SPLINE
SPL {X  -154.371, Y  +335.471, Z    +0.000, E1   +73.016, E3 +26676.206}
SPL {X  -149.938, Y  +321.685, Z    +0.000, E1   +73.398, E3 +26680.901}
SPL {X  -145.016, Y  +309.920, Z    +0.000, E1   +73.647, E3 +26685.422}
SPL {X  -139.138, Y  +298.522, Z    +0.000, E1   +74.138, E3 +26687.438}
SPL {X  -135.697, Y  +292.747, Z    +0.000, E1   +74.259, E3 +26689.439}
SPL {X  -132.590, Y  +287.964, Z    +0.000, E1   +73.910, E3 +26694.468}
SPL {X  -129.541, Y  +283.606, Z    +0.000, E1   +73.551, E3 +26699.108}
SPL {X  -126.457, Y  +279.493, Z    +0.000, E1   +73.175, E3 +26703.507}
SPL {X  -122.770, Y  +274.912, Z    +0.000, E1   +72.712, E3 +26708.362}
SPL {X  -118.941, Y  +270.496, Z    +0.000, E1   +72.188, E3 +26712.950}
SPL {X   -74.907, Y  +236.129, Z    +0.000, E1   +61.720, E3 +26791.563}
ENDSPLINE

SPLINE
SPL {X   -94.059, Y  +248.080, Z    +0.000, E1   +58.275, E3 +27013.256}
SPL {X  -136.558, Y  +294.141, Z    +0.000, E1   +54.887, E3 +27057.111}
SPL {X  -151.843, Y  +327.098, Z    +0.000, E1   +44.118, E3 +27066.470}
SPL {X  -157.484, Y  +349.293, Z    +0.000, E1   +30.654, E3 +27069.510}
SPL {X  -159.556, Y  +365.719, Z    +0.000, E1   +15.845, E3 +27070.702}
SPL {X  -159.982, Y  +375.924, Z    +0.000, E1    +4.476, E3 +27071.004}
SPL {X  -159.990, Y  +379.531, Z    +0.000, E1    -0.039, E3 +27071.031}
SPL {X  -159.990, Y  +382.420, Z    +0.000, E1    -7.600, E3 +27071.059}
SPL {X  -159.990, Y  +386.504, Z    +0.000, E1   -19.860, E3 +27071.165}
SPL {X  -159.990, Y  +392.530, Z    +0.000, E1   -36.133, E3 +27071.480}
SPL {X  -159.990, Y  +400.492, Z    +0.000, E1   -51.837, E3 +27072.133}
SPL {X  -159.990, Y  +409.662, Z    +0.000, E1   -61.705, E3 +27073.244}
SPL {X  -159.990, Y  +434.697, Z    +0.000, E1   -71.504, E3 +27078.264}
SPL {X  -159.990, Y  +521.523, Z    +0.000, E1   -76.035, E3 +27104.544}
SPL {X  -154.459, Y  +718.205, Z    +0.000, E1   -76.329, E3 +27186.340}
SPL {X  -151.356, Y  +728.349, Z    +0.000, E1   -76.056, E3 +27194.555}
SPL {X  -148.399, Y  +736.287, Z    +0.000, E1   -75.788, E3 +27201.434}
SPL {X  -144.005, Y  +746.209, Z    +0.000, E1   -75.396, E3 +27210.550}
SPL {X  -138.117, Y  +757.250, Z    +0.000, E1   -74.803, E3 +27221.440}
SPL {X  -133.491, Y  +764.686, Z    +0.000, E1   -74.276, E3 +27229.181}
SPL {X  -128.839, Y  +771.354, Z    +0.000, E1   -73.759, E3 +27236.199}
SPL {X  -123.568, Y  +778.125, Z    +0.000, E1   -73.105, E3 +27243.371}
SPL {X  -118.985, Y  +783.455, Z    +0.000, E1   -72.490, E3 +27248.879}
SPL {X   -72.391, Y  +819.176, Z    +0.000, E1   -59.867, E3 +27345.565}
ENDSPLINE

SPLINE
SPL {X   -92.809, Y  +806.820, Z    +0.000, E1   -56.994, E3 +27538.360}
SPL {X  -120.521, Y  +781.721, Z    +0.000, E1   -56.766, E3 +27574.459}
SPL {X  -148.710, Y  +735.509, Z    +0.000, E1   -46.282, E3 +27595.740}
SPL {X  -157.559, Y  +704.285, Z    +0.000, E1   -29.037, E3 +27601.069}
SPL {X  -159.430, Y  +689.871, Z    +0.000, E1   -16.582, E3 +27602.219}
SPL {X  -159.960, Y  +679.609, Z    +0.000, E1    -6.021, E3 +27602.602}
SPL {X  -159.990, Y  +674.508, Z    +0.000, E1    -0.018, E3 +27602.661}
SPL {X  -159.990, Y  +672.787, Z    +0.000, E1    +4.022, E3 +27602.673}
SPL {X  -159.990, Y  +669.267, Z    +0.000, E1   +13.665, E3 +27602.743}
SPL {X  -159.990, Y  +663.438, Z    +0.000, E1   +29.379, E3 +27603.014}
SPL {X  -159.990, Y  +655.264, Z    +0.000, E1   +47.291, E3 +27603.631}
SPL {X  -159.990, Y  +645.368, Z    +0.000, E1   +59.257, E3 +27604.874}
SPL {X  -159.990, Y  +624.023, Z    +0.000, E1   +69.513, E3 +27608.999}
SPL {X  -159.990, Y  +543.075, Z    +0.000, E1   +75.590, E3 +27632.647}
SPL {X  -156.121, Y  +342.530, Z    +0.000, E1   +75.868, E3 +27719.293}
SPL {X  -153.865, Y  +333.657, Z    +0.000, E1   +75.438, E3 +27728.897}
ENDSPLINE

SPLINE
SPL {X  -159.644, Y  +366.989, Z    +0.000, E1   +72.058, E3 +27744.424}
ENDSPLINE

SPLINE
SPL {X  -156.933, Y  +346.374, Z    +0.000, E1   +72.645, E3 +27752.313}
SPL {X  -151.144, Y  +325.039, Z    +0.000, E1   +73.323, E3 +27758.993}
SPL {X  -145.016, Y  +309.920, Z    +0.000, E1   +73.647, E3 +27764.787}
SPL {X  -136.944, Y  +294.777, Z    +0.000, E1   +74.219, E3 +27768.088}
SPL {X  -132.590, Y  +287.964, Z    +0.000, E1   +73.910, E3 +27773.833}
SPL {X  -129.541, Y  +283.606, Z    +0.000, E1   +73.551, E3 +27778.473}
SPL {X  -125.403, Y  +278.147, Z    +0.000, E1   +73.063, E3 +27784.280}
SPL {X  -121.908, Y  +273.889, Z    +0.000, E1   +72.578, E3 +27788.827}
SPL {X  -118.941, Y  +270.496, Z    +0.000, E1   +72.188, E3 +27792.315}
SPL {X   -74.907, Y  +236.129, Z    +0.000, E1   +61.720, E3 +27870.928}
ENDSPLINE

SPLINE
SPL {X   -94.059, Y  +248.080, Z    +0.000, E1   +58.275, E3 +28092.621}
SPL {X  -136.558, Y  +294.141, Z    +0.000, E1   +54.887, E3 +28136.476}
SPL {X  -151.843, Y  +327.098, Z    +0.000, E1   +44.118, E3 +28145.835}
SPL {X  -157.484, Y  +349.293, Z    +0.000, E1   +30.654, E3 +28148.875}
SPL {X  -159.556, Y  +365.719, Z    +0.000, E1   +15.845, E3 +28150.067}
SPL {X  -159.982, Y  +375.924, Z    +0.000, E1    +4.476, E3 +28150.369}
SPL {X  -159.990, Y  +379.531, Z    +0.000, E1    -0.039, E3 +28150.396}
SPL {X  -159.990, Y  +382.420, Z    +0.000, E1    -7.600, E3 +28150.424}
SPL {X  -159.990, Y  +386.504, Z    +0.000, E1   -19.860, E3 +28150.530}
SPL {X  -159.990, Y  +392.530, Z    +0.000, E1   -36.133, E3 +28150.845}
SPL {X  -159.990, Y  +400.492, Z    +0.000, E1   -51.837, E3 +28151.498}
SPL {X  -159.990, Y  +409.662, Z    +0.000, E1   -61.705, E3 +28152.609}
SPL {X  -159.990, Y  +434.697, Z    +0.000, E1   -71.504, E3 +28157.629}
SPL {X  -159.990, Y  +521.523, Z    +0.000, E1   -76.035, E3 +28183.909}
SPL {X  -154.459, Y  +718.205, Z    +0.000, E1   -76.329, E3 +28265.705}
SPL {X  -151.356, Y  +728.349, Z    +0.000, E1   -76.056, E3 +28273.920}
SPL {X  -148.399, Y  +736.287, Z    +0.000, E1   -75.788, E3 +28280.799}
SPL {X  -144.005, Y  +746.209, Z    +0.000, E1   -75.396, E3 +28289.915}
SPL {X  -138.117, Y  +757.250, Z    +0.000, E1   -74.803, E3 +28300.805}
SPL {X  -133.491, Y  +764.686, Z    +0.000, E1   -74.276, E3 +28308.546}
SPL {X  -130.530, Y  +769.013, Z    +0.000, E1   -73.929, E3 +28313.128}
SPL {X  -127.734, Y  +772.837, Z    +0.000, E1   -73.601, E3 +28317.180}
SPL {X  -124.765, Y  +776.652, Z    +0.000, E1   -73.233, E3 +28321.214}
SPL {X  -121.376, Y  +780.734, Z    +0.000, E1   -72.804, E3 +28325.476}
SPL {X  -118.281, Y  +784.233, Z    +0.000, E1   -72.371, E3 +28329.044}
SPL {X   -72.391, Y  +819.176, Z    +0.000, E1   -59.867, E3 +28424.930}
ENDSPLINE

SPLINE
SPL {X   -92.809, Y  +806.820, Z    +0.000, E1   -56.994, E3 +28617.725}
SPL {X  -120.521, Y  +781.721, Z    +0.000, E1   -56.766, E3 +28653.824}
SPL {X  -148.710, Y  +735.509, Z    +0.000, E1   -46.282, E3 +28675.105}
SPL {X  -157.559, Y  +704.285, Z    +0.000, E1   -29.037, E3 +28680.434}
SPL {X  -159.430, Y  +689.871, Z    +0.000, E1   -16.582, E3 +28681.584}
SPL {X  -159.960, Y  +679.609, Z    +0.000, E1    -6.021, E3 +28681.968}
SPL {X  -159.990, Y  +674.508, Z    +0.000, E1    -0.018, E3 +28682.026}
SPL {X  -159.990, Y  +672.787, Z    +0.000, E1    +4.022, E3 +28682.038}
SPL {X  -159.990, Y  +669.267, Z    +0.000, E1   +13.665, E3 +28682.108}
SPL {X  -159.990, Y  +665.069, Z    +0.000, E1   +25.376, E3 +28682.280}
SPL {X  -159.990, Y  +657.821, Z    +0.000, E1   +42.408, E3 +28682.782}
SPL {X  -159.990, Y  +645.368, Z    +0.000, E1   +59.257, E3 +28684.239}
SPL {X  -159.990, Y  +624.023, Z    +0.000, E1   +69.513, E3 +28688.364}
SPL {X  -159.990, Y  +543.075, Z    +0.000, E1   +75.590, E3 +28712.012}
SPL {X  -156.121, Y  +342.530, Z    +0.000, E1   +75.868, E3 +28798.658}
SPL {X  -153.498, Y  +332.386, Z    +0.000, E1   +75.628, E3 +28806.663}
ENDSPLINE

SPLINE
SPL {X  -155.252, Y  +338.851, Z    +0.000, E1   +74.632, E3 +28814.041}
SPL {X  -159.644, Y  +366.989, Z    +0.000, E1   +72.058, E3 +28823.789}
ENDSPLINE

SPLINE
SPL {X  -156.933, Y  +346.374, Z    +0.000, E1   +72.645, E3 +28831.678}
SPL {X  -151.144, Y  +325.039, Z    +0.000, E1   +73.323, E3 +28838.358}
SPL {X  -146.668, Y  +313.584, Z    +0.000, E1   +73.560, E3 +28842.840}
SPL {X  -141.230, Y  +302.327, Z    +0.000, E1   +73.933, E3 +28845.811}
SPL {X  -135.697, Y  +292.747, Z    +0.000, E1   +74.259, E3 +28848.170}
SPL {X  -132.590, Y  +287.964, Z    +0.000, E1   +73.910, E3 +28853.198}
SPL {X  -129.541, Y  +283.606, Z    +0.000, E1   +73.551, E3 +28857.838}
SPL {X  -125.403, Y  +278.147, Z    +0.000, E1   +73.063, E3 +28863.645}
SPL {X  -121.908, Y  +273.889, Z    +0.000, E1   +72.578, E3 +28868.192}
SPL {X  -118.941, Y  +270.496, Z    +0.000, E1   +72.188, E3 +28871.680}
SPL {X   -74.907, Y  +236.129, Z    +0.000, E1   +61.720, E3 +28950.293}
SPL {X   -72.759, Y  +235.012, Z    +0.000, E1   +56.036, E3 +29121.971}
ENDSPLINE

SPLINE
SPL {X  -123.257, Y  +275.497, Z    +0.000, E1   +57.800, E3 +29205.847}
SPL {X  -149.689, Y  +321.019, Z    +0.000, E1   +46.817, E3 +29223.947}
SPL {X  -157.484, Y  +349.293, Z    +0.000, E1   +30.654, E3 +29228.240}
SPL {X  -159.556, Y  +365.719, Z    +0.000, E1   +15.845, E3 +29229.432}
SPL {X  -159.982, Y  +375.924, Z    +0.000, E1    +4.476, E3 +29229.734}
SPL {X  -159.990, Y  +379.531, Z    +0.000, E1    -0.039, E3 +29229.761}
SPL {X  -159.990, Y  +382.420, Z    +0.000, E1    -7.600, E3 +29229.789}
SPL {X  -159.990, Y  +387.978, Z    +0.000, E1   -23.882, E3 +29229.958}
SPL {X  -159.990, Y  +396.850, Z    +0.000, E1   -45.459, E3 +29230.545}
SPL {X  -159.990, Y  +409.662, Z    +0.000, E1   -61.705, E3 +29231.974}
SPL {X  -159.990, Y  +426.583, Z    +0.000, E1   -69.729, E3 +29235.088}
SPL {X  -159.990, Y  +451.842, Z    +0.000, E1   -73.935, E3 +29241.015}
SPL {X  -159.990, Y  +521.523, Z    +0.000, E1   -76.035, E3 +29263.275}
SPL {X  -154.459, Y  +718.205, Z    +0.000, E1   -76.329, E3 +29345.070}
SPL {X  -151.356, Y  +728.349, Z    +0.000, E1   -76.056, E3 +29353.285}
SPL {X  -148.399, Y  +736.287, Z    +0.000, E1   -75.788, E3 +29360.164}
SPL {X  -144.005, Y  +746.209, Z    +0.000, E1   -75.396, E3 +29369.280}
SPL {X  -138.117, Y  +757.250, Z    +0.000, E1   -74.803, E3 +29380.170}
SPL {X  -133.491, Y  +764.686, Z    +0.000, E1   -74.276, E3 +29387.911}
SPL {X  -130.530, Y  +769.013, Z    +0.000, E1   -73.929, E3 +29392.493}
SPL {X  -127.734, Y  +772.837, Z    +0.000, E1   -73.601, E3 +29396.545}
SPL {X  -123.568, Y  +778.125, Z    +0.000, E1   -73.105, E3 +29402.101}
SPL {X  -118.985, Y  +783.455, Z    +0.000, E1   -72.490, E3 +29407.609}
SPL {X   -72.391, Y  +819.176, Z    +0.000, E1   -59.867, E3 +29504.295}
ENDSPLINE

SPLINE
SPL {X  -116.241, Y  +786.431, Z    +0.000, E1   -57.120, E3 +29728.737}
SPL {X  -148.710, Y  +735.509, Z    +0.000, E1   -46.282, E3 +29754.470}
SPL {X  -156.039, Y  +711.834, Z    +0.000, E1   -34.227, E3 +29758.955}
SPL {X  -158.281, Y  +699.823, Z    +0.000, E1   -25.469, E3 +29760.246}
SPL {X  -159.709, Y  +685.986, Z    +0.000, E1   -12.810, E3 +29761.131}
SPL {X  -159.990, Y  +674.648, Z    +0.000, E1    -0.349, E3 +29761.390}
SPL {X  -159.990, Y  +672.787, Z    +0.000, E1    +4.022, E3 +29761.403}
SPL {X  -159.990, Y  +669.267, Z    +0.000, E1   +13.665, E3 +29761.473}
SPL {X  -159.990, Y  +665.069, Z    +0.000, E1   +25.376, E3 +29761.645}
SPL {X  -159.990, Y  +657.821, Z    +0.000, E1   +42.408, E3 +29762.147}
SPL {X  -159.990, Y  +645.368, Z    +0.000, E1   +59.257, E3 +29763.604}
SPL {X  -159.990, Y  +624.023, Z    +0.000, E1   +69.513, E3 +29767.729}
SPL {X  -159.990, Y  +543.075, Z    +0.000, E1   +75.590, E3 +29791.377}
SPL {X  -156.121, Y  +342.530, Z    +0.000, E1   +75.868, E3 +29878.023}
SPL {X  -153.498, Y  +332.386, Z    +0.000, E1   +75.628, E3 +29886.028}
ENDSPLINE

SPLINE
SPL {X  -155.252, Y  +338.851, Z    +0.000, E1   +74.632, E3 +29893.406}
SPL {X  -159.103, Y  +360.678, Z    +0.000, E1   +72.233, E3 +29905.731}
ENDSPLINE

SPLINE
SPL {X  -154.371, Y  +335.471, Z    +0.000, E1   +73.016, E3 +29914.302}
SPL {X  -149.938, Y  +321.685, Z    +0.000, E1   +73.398, E3 +29918.996}
SPL {X  -145.016, Y  +309.920, Z    +0.000, E1   +73.647, E3 +29923.517}
SPL {X  -139.138, Y  +298.522, Z    +0.000, E1   +74.138, E3 +29925.533}
SPL {X  -135.697, Y  +292.747, Z    +0.000, E1   +74.259, E3 +29927.535}
SPL {X  -132.590, Y  +287.964, Z    +0.000, E1   +73.910, E3 +29932.563}
SPL {X  -129.541, Y  +283.606, Z    +0.000, E1   +73.551, E3 +29937.203}
SPL {X  -126.457, Y  +279.493, Z    +0.000, E1   +73.175, E3 +29941.602}
SPL {X  -122.770, Y  +274.912, Z    +0.000, E1   +72.712, E3 +29946.458}
SPL {X  -119.156, Y  +270.736, Z    +0.000, E1   +72.213, E3 +29950.807}
SPL {X  -117.531, Y  +268.949, Z    +0.000, E1   +71.964, E3 +29952.622}
SPL {X   -74.907, Y  +236.129, Z    +0.000, E1   +61.720, E3 +30029.658}
ENDSPLINE

SPLINE
SPL {X   -94.059, Y  +248.080, Z    +0.000, E1   +58.275, E3 +30251.351}
SPL {X  -130.769, Y  +285.325, Z    +0.000, E1   +56.495, E3 +30291.228}
SPL {X  -149.689, Y  +321.019, Z    +0.000, E1   +46.817, E3 +30303.312}
SPL {X  -157.484, Y  +349.293, Z    +0.000, E1   +30.654, E3 +30307.605}
SPL {X  -159.556, Y  +365.719, Z    +0.000, E1   +15.845, E3 +30308.797}
SPL {X  -159.982, Y  +375.924, Z    +0.000, E1    +4.476, E3 +30309.099}
SPL {X  -159.990, Y  +379.531, Z    +0.000, E1    -0.039, E3 +30309.126}
SPL {X  -159.990, Y  +382.420, Z    +0.000, E1    -7.600, E3 +30309.154}
SPL {X  -159.990, Y  +386.504, Z    +0.000, E1   -19.860, E3 +30309.260}
SPL {X  -159.990, Y  +392.530, Z    +0.000, E1   -36.133, E3 +30309.575}
SPL {X  -159.990, Y  +400.492, Z    +0.000, E1   -51.837, E3 +30310.228}
SPL {X  -159.990, Y  +409.662, Z    +0.000, E1   -61.705, E3 +30311.339}
SPL {X  -159.990, Y  +434.697, Z    +0.000, E1   -71.504, E3 +30316.359}
SPL {X  -159.990, Y  +521.523, Z    +0.000, E1   -76.035, E3 +30342.640}
SPL {X  -154.459, Y  +718.205, Z    +0.000, E1   -76.329, E3 +30424.435}
SPL {X  -151.356, Y  +728.349, Z    +0.000, E1   -76.056, E3 +30432.650}
SPL {X  -148.399, Y  +736.287, Z    +0.000, E1   -75.788, E3 +30439.529}
SPL {X  -144.005, Y  +746.209, Z    +0.000, E1   -75.396, E3 +30448.645}
SPL {X  -138.117, Y  +757.250, Z    +0.000, E1   -74.803, E3 +30459.535}
SPL {X  -133.491, Y  +764.686, Z    +0.000, E1   -74.276, E3 +30467.276}
SPL {X  -128.839, Y  +771.354, Z    +0.000, E1   -73.759, E3 +30474.295}
SPL {X  -123.568, Y  +778.125, Z    +0.000, E1   -73.105, E3 +30481.466}
SPL {X  -118.985, Y  +783.455, Z    +0.000, E1   -72.490, E3 +30486.974}
SPL {X   -72.391, Y  +819.176, Z    +0.000, E1   -59.867, E3 +30583.660}
ENDSPLINE

SPLINE
SPL {X   -92.809, Y  +806.820, Z    +0.000, E1   -56.994, E3 +30776.455}
SPL {X  -120.521, Y  +781.721, Z    +0.000, E1   -56.766, E3 +30812.554}
SPL {X  -148.710, Y  +735.509, Z    +0.000, E1   -46.282, E3 +30833.835}
SPL {X  -157.559, Y  +704.285, Z    +0.000, E1   -29.037, E3 +30839.164}
SPL {X  -159.430, Y  +689.871, Z    +0.000, E1   -16.582, E3 +30840.315}
SPL {X  -159.960, Y  +679.609, Z    +0.000, E1    -6.021, E3 +30840.698}
SPL {X  -159.990, Y  +674.508, Z    +0.000, E1    -0.018, E3 +30840.756}
SPL {X  -159.990, Y  +672.787, Z    +0.000, E1    +4.022, E3 +30840.768}
SPL {X  -159.990, Y  +669.267, Z    +0.000, E1   +13.665, E3 +30840.838}
SPL {X  -159.990, Y  +663.438, Z    +0.000, E1   +29.379, E3 +30841.109}
SPL {X  -159.990, Y  +655.264, Z    +0.000, E1   +47.291, E3 +30841.726}
SPL {X  -159.990, Y  +645.368, Z    +0.000, E1   +59.257, E3 +30842.969}
SPL {X  -159.990, Y  +624.023, Z    +0.000, E1   +69.513, E3 +30847.094}
SPL {X  -159.990, Y  +543.075, Z    +0.000, E1   +75.590, E3 +30870.742}
SPL {X  -156.121, Y  +342.530, Z    +0.000, E1   +75.868, E3 +30957.388}
SPL {X  -153.865, Y  +333.657, Z    +0.000, E1   +75.438, E3 +30966.992}
ENDSPLINE

SPLINE
SPL {X  -159.103, Y  +360.678, Z    +0.000, E1   +72.233, E3 +30985.096}
ENDSPLINE

SPLINE
SPL {X  -154.371, Y  +335.471, Z    +0.000, E1   +73.016, E3 +30993.667}
SPL {X  -148.318, Y  +317.512, Z    +0.000, E1   +73.488, E3 +30999.988}
SPL {X  -141.230, Y  +302.327, Z    +0.000, E1   +73.933, E3 +31004.541}
SPL {X  -135.697, Y  +292.747, Z    +0.000, E1   +74.259, E3 +31006.900}
SPL {X  -132.590, Y  +287.964, Z    +0.000, E1   +73.910, E3 +31011.928}
SPL {X  -129.541, Y  +283.606, Z    +0.000, E1   +73.551, E3 +31016.568}
SPL {X  -126.457, Y  +279.493, Z    +0.000, E1   +73.175, E3 +31020.967}
SPL {X  -122.770, Y  +274.912, Z    +0.000, E1   +72.712, E3 +31025.823}
SPL {X  -119.156, Y  +270.736, Z    +0.000, E1   +72.213, E3 +31030.172}
SPL {X  -117.531, Y  +268.949, Z    +0.000, E1   +71.964, E3 +31031.988}
SPL {X   -74.907, Y  +236.129, Z    +0.000, E1   +61.720, E3 +31109.024}
SPL {X   -72.759, Y  +235.012, Z    +0.000, E1   +56.036, E3 +31280.701}
ENDSPLINE

SPLINE
SPL {X  -110.316, Y  +261.624, Z    +0.000, E1   +58.739, E3 +31352.774}
SPL {X  -136.558, Y  +294.141, Z    +0.000, E1   +54.887, E3 +31374.571}
SPL {X  -153.807, Y  +333.452, Z    +0.000, E1   +40.945, E3 +31384.968}
SPL {X  -158.168, Y  +353.421, Z    +0.000, E1   +27.296, E3 +31387.361}
SPL {X  -159.556, Y  +365.719, Z    +0.000, E1   +15.845, E3 +31388.162}
SPL {X  -159.982, Y  +375.924, Z    +0.000, E1    +4.476, E3 +31388.464}
SPL {X  -159.990, Y  +379.800, Z    +0.000, E1    -0.377, E3 +31388.493}
SPL {X  -159.990, Y  +383.422, Z    +0.000, E1   -10.730, E3 +31388.536}
SPL {X  -159.990, Y  +387.978, Z    +0.000, E1   -23.882, E3 +31388.688}
SPL {X  -159.990, Y  +394.494, Z    +0.000, E1   -40.961, E3 +31389.069}
SPL {X  -159.990, Y  +400.492, Z    +0.000, E1   -51.837, E3 +31389.593}
SPL {X  -159.990, Y  +409.662, Z    +0.000, E1   -61.705, E3 +31390.704}
SPL {X  -159.990, Y  +434.697, Z    +0.000, E1   -71.504, E3 +31395.724}
SPL {X  -159.990, Y  +521.523, Z    +0.000, E1   -76.035, E3 +31422.005}
SPL {X  -154.459, Y  +718.205, Z    +0.000, E1   -76.329, E3 +31503.800}
SPL {X  -151.356, Y  +728.349, Z    +0.000, E1   -76.056, E3 +31512.016}
SPL {X  -147.124, Y  +739.360, Z    +0.000, E1   -75.690, E3 +31521.612}
SPL {X  -142.861, Y  +748.524, Z    +0.000, E1   -75.261, E3 +31530.297}
SPL {X  -139.796, Y  +754.307, Z    +0.000, E1   -74.951, E3 +31535.985}
SPL {X  -136.850, Y  +759.378, Z    +0.000, E1   -74.643, E3 +31541.129}
SPL {X  -133.491, Y  +764.686, Z    +0.000, E1   -74.276, E3 +31546.641}
SPL {X  -128.839, Y  +771.354, Z    +0.000, E1   -73.759, E3 +31553.660}
SPL {X  -124.765, Y  +776.652, Z    +0.000, E1   -73.233, E3 +31559.310}
SPL {X  -121.376, Y  +780.734, Z    +0.000, E1   -72.804, E3 +31563.571}
SPL {X  -118.281, Y  +784.233, Z    +0.000, E1   -72.371, E3 +31567.140}
SPL {X   -72.391, Y  +819.176, Z    +0.000, E1   -59.867, E3 +31663.025}
ENDSPLINE

SPLINE
SPL {X  -116.241, Y  +786.431, Z    +0.000, E1   -57.120, E3 +31887.468}
SPL {X  -143.482, Y  +747.279, Z    +0.000, E1   -50.227, E3 +31909.932}
SPL {X  -154.118, Y  +719.449, Z    +0.000, E1   -38.836, E3 +31916.511}
SPL {X  -158.958, Y  +694.646, Z    +0.000, E1   -21.132, E3 +31919.363}
SPL {X  -159.960, Y  +679.609, Z    +0.000, E1    -6.021, E3 +31920.063}
SPL {X  -159.990, Y  +674.508, Z    +0.000, E1    -0.018, E3 +31920.121}
SPL {X  -159.990, Y  +672.787, Z    +0.000, E1    +4.022, E3 +31920.133}
SPL {X  -159.990, Y  +669.267, Z    +0.000, E1   +13.665, E3 +31920.203}
SPL {X  -159.990, Y  +665.069, Z    +0.000, E1   +25.376, E3 +31920.375}
SPL {X  -159.990, Y  +657.821, Z    +0.000, E1   +42.408, E3 +31920.878}
SPL {X  -159.990, Y  +645.368, Z    +0.000, E1   +59.257, E3 +31922.334}
SPL {X  -159.990, Y  +624.023, Z    +0.000, E1   +69.513, E3 +31926.459}
SPL {X  -159.990, Y  +543.075, Z    +0.000, E1   +75.590, E3 +31950.107}
SPL {X  -156.121, Y  +342.530, Z    +0.000, E1   +75.868, E3 +32036.753}
SPL {X  -153.865, Y  +333.657, Z    +0.000, E1   +75.438, E3 +32046.357}
ENDSPLINE

SPLINE
SPL {X  -159.644, Y  +366.989, Z    +0.000, E1   +72.058, E3 +32061.884}
ENDSPLINE

SPLINE
SPL {X  -156.933, Y  +346.374, Z    +0.000, E1   +72.645, E3 +32069.774}
SPL {X  -151.144, Y  +325.039, Z    +0.000, E1   +73.323, E3 +32076.453}
SPL {X  -145.016, Y  +309.920, Z    +0.000, E1   +73.647, E3 +32082.247}
SPL {X  -136.944, Y  +294.777, Z    +0.000, E1   +74.219, E3 +32085.549}
SPL {X  -132.590, Y  +287.964, Z    +0.000, E1   +73.910, E3 +32091.293}
SPL {X  -129.541, Y  +283.606, Z    +0.000, E1   +73.551, E3 +32095.934}
SPL {X  -125.403, Y  +278.147, Z    +0.000, E1   +73.063, E3 +32101.741}
SPL {X  -121.908, Y  +273.889, Z    +0.000, E1   +72.578, E3 +32106.287}
SPL {X  -118.941, Y  +270.496, Z    +0.000, E1   +72.188, E3 +32109.775}
SPL {X   -74.907, Y  +236.129, Z    +0.000, E1   +61.720, E3 +32188.389}
ENDSPLINE

SPLINE
SPL {X   -94.059, Y  +248.080, Z    +0.000, E1   +58.275, E3 +32410.082}
SPL {X  -136.558, Y  +294.141, Z    +0.000, E1   +54.887, E3 +32453.936}
SPL {X  -151.843, Y  +327.098, Z    +0.000, E1   +44.118, E3 +32463.296}
SPL {X  -157.484, Y  +349.293, Z    +0.000, E1   +30.654, E3 +32466.335}
SPL {X  -159.556, Y  +365.719, Z    +0.000, E1   +15.845, E3 +32467.528}
SPL {X  -159.982, Y  +375.924, Z    +0.000, E1    +4.476, E3 +32467.829}
SPL {X  -159.990, Y  +379.531, Z    +0.000, E1    -0.039, E3 +32467.856}
SPL {X  -159.990, Y  +382.420, Z    +0.000, E1    -7.600, E3 +32467.885}
SPL {X  -159.990, Y  +387.978, Z    +0.000, E1   -23.882, E3 +32468.053}
SPL {X  -159.990, Y  +396.850, Z    +0.000, E1   -45.459, E3 +32468.640}
SPL {X  -159.990, Y  +409.662, Z    +0.000, E1   -61.705, E3 +32470.069}
SPL {X  -159.990, Y  +426.583, Z    +0.000, E1   -69.729, E3 +32473.183}
SPL {X  -159.990, Y  +451.842, Z    +0.000, E1   -73.935, E3 +32479.110}
SPL {X  -159.990, Y  +521.523, Z    +0.000, E1   -76.035, E3 +32501.370}
SPL {X  -154.459, Y  +718.205, Z    +0.000, E1   -76.329, E3 +32583.165}
SPL {X  -151.356, Y  +728.349, Z    +0.000, E1   -76.056, E3 +32591.381}
SPL {X  -148.399, Y  +736.287, Z    +0.000, E1   -75.788, E3 +32598.259}
SPL {X  -144.005, Y  +746.209, Z    +0.000, E1   -75.396, E3 +32607.375}
SPL {X  -138.117, Y  +757.250, Z    +0.000, E1   -74.803, E3 +32618.265}
SPL {X  -133.491, Y  +764.686, Z    +0.000, E1   -74.276, E3 +32626.006}
SPL {X  -130.530, Y  +769.013, Z    +0.000, E1   -73.929, E3 +32630.588}
SPL {X  -127.734, Y  +772.837, Z    +0.000, E1   -73.601, E3 +32634.640}
SPL {X  -124.765, Y  +776.652, Z    +0.000, E1   -73.233, E3 +32638.675}
SPL {X  -121.376, Y  +780.734, Z    +0.000, E1   -72.804, E3 +32642.936}
SPL {X  -118.281, Y  +784.233, Z    +0.000, E1   -72.371, E3 +32646.505}
SPL {X   -72.391, Y  +819.176, Z    +0.000, E1   -59.867, E3 +32742.390}
ENDSPLINE

SPLINE
SPL {X  -116.241, Y  +786.431, Z    +0.000, E1   -57.120, E3 +32966.833}
SPL {X  -148.710, Y  +735.509, Z    +0.000, E1   -46.282, E3 +32992.565}
SPL {X  -157.559, Y  +704.285, Z    +0.000, E1   -29.037, E3 +32997.895}
SPL {X  -159.709, Y  +685.986, Z    +0.000, E1   -12.810, E3 +32999.226}
SPL {X  -159.990, Y  +674.648, Z    +0.000, E1    -0.349, E3 +32999.486}
SPL {X  -159.990, Y  +672.787, Z    +0.000, E1    +4.022, E3 +32999.498}
SPL {X  -159.990, Y  +669.267, Z    +0.000, E1   +13.665, E3 +32999.569}
SPL {X  -159.990, Y  +663.438, Z    +0.000, E1   +29.379, E3 +32999.839}
SPL {X  -159.990, Y  +655.264, Z    +0.000, E1   +47.291, E3 +33000.456}
SPL {X  -159.990, Y  +645.368, Z    +0.000, E1   +59.257, E3 +33001.699}
SPL {X  -159.990, Y  +624.023, Z    +0.000, E1   +69.513, E3 +33005.824}
SPL {X  -159.990, Y  +543.075, Z    +0.000, E1   +75.590, E3 +33029.472}
SPL {X  -156.121, Y  +342.530, Z    +0.000, E1   +75.868, E3 +33116.118}
SPL {X  -153.498, Y  +332.386, Z    +0.000, E1   +75.628, E3 +33124.123}
ENDSPLINE

SPLINE
SPL {X  -155.252, Y  +338.851, Z    +0.000, E1   +74.632, E3 +33131.501}
SPL {X  -159.103, Y  +360.678, Z    +0.000, E1   +72.233, E3 +33143.826}
ENDSPLINE

SPLINE
SPL {X  -154.371, Y  +335.471, Z    +0.000, E1   +73.016, E3 +33152.397}
SPL {X  -149.938, Y  +321.685, Z    +0.000, E1   +73.398, E3 +33157.091}
SPL {X  -145.016, Y  +309.920, Z    +0.000, E1   +73.647, E3 +33161.612}
SPL {X  -136.944, Y  +294.777, Z    +0.000, E1   +74.219, E3 +33164.914}
SPL {X  -132.590, Y  +287.964, Z    +0.000, E1   +73.910, E3 +33170.658}
SPL {X  -129.541, Y  +283.606, Z    +0.000, E1   +73.551, E3 +33175.299}
SPL {X  -125.403, Y  +278.147, Z    +0.000, E1   +73.063, E3 +33181.106}
SPL {X  -121.908, Y  +273.889, Z    +0.000, E1   +72.578, E3 +33185.652}
SPL {X  -119.156, Y  +270.736, Z    +0.000, E1   +72.213, E3 +33188.902}
SPL {X  -117.531, Y  +268.949, Z    +0.000, E1   +71.964, E3 +33190.718}
SPL {X   -74.907, Y  +236.129, Z    +0.000, E1   +61.720, E3 +33267.754}
ENDSPLINE

SPLINE
SPL {X   -94.059, Y  +248.080, Z    +0.000, E1   +58.275, E3 +33489.447}
SPL {X  -130.769, Y  +285.325, Z    +0.000, E1   +56.495, E3 +33529.324}
SPL {X  -149.689, Y  +321.019, Z    +0.000, E1   +46.817, E3 +33541.408}
SPL {X  -157.484, Y  +349.293, Z    +0.000, E1   +30.654, E3 +33545.700}
SPL {X  -159.556, Y  +365.719, Z    +0.000, E1   +15.845, E3 +33546.893}
SPL {X  -159.982, Y  +375.924, Z    +0.000, E1    +4.476, E3 +33547.194}
SPL {X  -159.990, Y  +379.531, Z    +0.000, E1    -0.039, E3 +33547.221}
SPL {X  -159.990, Y  +382.420, Z    +0.000, E1    -7.600, E3 +33547.250}
SPL {X  -159.990, Y  +386.504, Z    +0.000, E1   -19.860, E3 +33547.355}
SPL {X  -159.990, Y  +392.530, Z    +0.000, E1   -36.133, E3 +33547.670}
SPL {X  -159.990, Y  +400.492, Z    +0.000, E1   -51.837, E3 +33548.323}
SPL {X  -159.990, Y  +409.662, Z    +0.000, E1   -61.705, E3 +33549.434}
SPL {X  -159.990, Y  +434.697, Z    +0.000, E1   -71.504, E3 +33554.454}
SPL {X  -159.990, Y  +521.523, Z    +0.000, E1   -76.035, E3 +33580.735}
SPL {X  -154.459, Y  +718.205, Z    +0.000, E1   -76.329, E3 +33662.530}
SPL {X  -151.356, Y  +728.349, Z    +0.000, E1   -76.056, E3 +33670.746}
SPL {X  -148.399, Y  +736.287, Z    +0.000, E1   -75.788, E3 +33677.624}
SPL {X  -144.005, Y  +746.209, Z    +0.000, E1   -75.396, E3 +33686.740}
SPL {X  -138.117, Y  +757.250, Z    +0.000, E1   -74.803, E3 +33697.630}
SPL {X  -133.491, Y  +764.686, Z    +0.000, E1   -74.276, E3 +33705.371}
SPL {X  -130.530, Y  +769.013, Z    +0.000, E1   -73.929, E3 +33709.953}
SPL {X  -127.734, Y  +772.837, Z    +0.000, E1   -73.601, E3 +33714.005}
SPL {X  -124.765, Y  +776.652, Z    +0.000, E1   -73.233, E3 +33718.040}
SPL {X  -121.376, Y  +780.734, Z    +0.000, E1   -72.804, E3 +33722.301}
SPL {X  -118.281, Y  +784.233, Z    +0.000, E1   -72.371, E3 +33725.870}
SPL {X   -72.391, Y  +819.176, Z    +0.000, E1   -59.867, E3 +33821.755}
ENDSPLINE

SPLINE
SPL {X  -116.241, Y  +786.431, Z    +0.000, E1   -57.120, E3 +34046.198}
SPL {X  -148.710, Y  +735.509, Z    +0.000, E1   -46.282, E3 +34071.930}
SPL {X  -157.559, Y  +704.285, Z    +0.000, E1   -29.037, E3 +34077.260}
SPL {X  -159.709, Y  +685.986, Z    +0.000, E1   -12.810, E3 +34078.591}
SPL {X  -159.990, Y  +674.648, Z    +0.000, E1    -0.349, E3 +34078.851}
SPL {X  -159.990, Y  +672.787, Z    +0.000, E1    +4.022, E3 +34078.863}
SPL {X  -159.990, Y  +669.267, Z    +0.000, E1   +13.665, E3 +34078.934}
SPL {X  -159.990, Y  +663.438, Z    +0.000, E1   +29.379, E3 +34079.204}
SPL {X  -159.990, Y  +655.264, Z    +0.000, E1   +47.291, E3 +34079.821}
SPL {X  -159.990, Y  +645.368, Z    +0.000, E1   +59.257, E3 +34081.064}
SPL {X  -159.990, Y  +624.023, Z    +0.000, E1   +69.513, E3 +34085.189}
SPL {X  -159.990, Y  +543.075, Z    +0.000, E1   +75.590, E3 +34108.837}
SPL {X  -156.121, Y  +342.530, Z    +0.000, E1   +75.868, E3 +34195.483}
SPL {X  -153.498, Y  +332.386, Z    +0.000, E1   +75.628, E3 +34203.488}
ENDSPLINE

SPLINE
SPL {X  -155.252, Y  +338.851, Z    +0.000, E1   +74.632, E3 +34210.866}
SPL {X  -159.103, Y  +360.678, Z    +0.000, E1   +72.233, E3 +34223.191}
ENDSPLINE

SPLINE
SPL {X  -154.371, Y  +335.471, Z    +0.000, E1   +73.016, E3 +34231.762}
SPL {X  -149.938, Y  +321.685, Z    +0.000, E1   +73.398, E3 +34236.456}
SPL {X  -145.016, Y  +309.920, Z    +0.000, E1   +73.647, E3 +34240.977}
SPL {X  -136.944, Y  +294.777, Z    +0.000, E1   +74.219, E3 +34244.279}
SPL {X  -132.590, Y  +287.964, Z    +0.000, E1   +73.910, E3 +34250.023}
SPL {X  -129.541, Y  +283.606, Z    +0.000, E1   +73.551, E3 +34254.664}
SPL {X  -125.403, Y  +278.147, Z    +0.000, E1   +73.063, E3 +34260.471}
SPL {X  -121.908, Y  +273.889, Z    +0.000, E1   +72.578, E3 +34265.017}
SPL {X  -119.156, Y  +270.736, Z    +0.000, E1   +72.213, E3 +34268.267}
SPL {X  -117.531, Y  +268.949, Z    +0.000, E1   +71.964, E3 +34270.083}
SPL {X   -74.907, Y  +236.129, Z    +0.000, E1   +61.720, E3 +34347.119}
ENDSPLINE

SPLINE
SPL {X   -94.059, Y  +248.080, Z    +0.000, E1   +58.275, E3 +34568.812}
SPL {X  -130.769, Y  +285.325, Z    +0.000, E1   +56.495, E3 +34608.689}
SPL {X  -149.689, Y  +321.019, Z    +0.000, E1   +46.817, E3 +34620.773}
SPL {X  -157.484, Y  +349.293, Z    +0.000, E1   +30.654, E3 +34625.065}
SPL {X  -159.556, Y  +365.719, Z    +0.000, E1   +15.845, E3 +34626.258}
SPL {X  -159.982, Y  +375.924, Z    +0.000, E1    +4.476, E3 +34626.559}
SPL {X  -159.990, Y  +379.531, Z    +0.000, E1    -0.039, E3 +34626.586}
SPL {X  -159.990, Y  +382.420, Z    +0.000, E1    -7.600, E3 +34626.615}
SPL {X  -159.990, Y  +386.504, Z    +0.000, E1   -19.860, E3 +34626.720}
SPL {X  -159.990, Y  +392.530, Z    +0.000, E1   -36.133, E3 +34627.035}
SPL {X  -159.990, Y  +400.492, Z    +0.000, E1   -51.837, E3 +34627.688}
SPL {X  -159.990, Y  +409.662, Z    +0.000, E1   -61.705, E3 +34628.799}
SPL {X  -159.990, Y  +434.697, Z    +0.000, E1   -71.504, E3 +34633.819}
SPL {X  -159.990, Y  +521.523, Z    +0.000, E1   -76.035, E3 +34660.100}
SPL {X  -154.459, Y  +718.205, Z    +0.000, E1   -76.329, E3 +34741.895}
SPL {X  -151.356, Y  +728.349, Z    +0.000, E1   -76.056, E3 +34750.111}
SPL {X  -148.399, Y  +736.287, Z    +0.000, E1   -75.788, E3 +34756.989}
SPL {X  -144.005, Y  +746.209, Z    +0.000, E1   -75.396, E3 +34766.105}
SPL {X  -138.117, Y  +757.250, Z    +0.000, E1   -74.803, E3 +34776.995}
SPL {X  -133.491, Y  +764.686, Z    +0.000, E1   -74.276, E3 +34784.736}
SPL {X  -130.530, Y  +769.013, Z    +0.000, E1   -73.929, E3 +34789.318}
SPL {X  -127.734, Y  +772.837, Z    +0.000, E1   -73.601, E3 +34793.370}
SPL {X  -124.765, Y  +776.652, Z    +0.000, E1   -73.233, E3 +34797.405}
SPL {X  -121.376, Y  +780.734, Z    +0.000, E1   -72.804, E3 +34801.666}
SPL {X  -118.281, Y  +784.233, Z    +0.000, E1   -72.371, E3 +34805.235}
SPL {X   -72.391, Y  +819.176, Z    +0.000, E1   -59.867, E3 +34901.120}
ENDSPLINE

SPLINE
SPL {X   -92.809, Y  +806.820, Z    +0.000, E1   -56.994, E3 +35093.916}
SPL {X  -120.521, Y  +781.721, Z    +0.000, E1   -56.766, E3 +35130.014}
SPL {X  -143.482, Y  +747.279, Z    +0.000, E1   -50.227, E3 +35148.027}
SPL {X  -154.118, Y  +719.449, Z    +0.000, E1   -38.836, E3 +35154.607}
SPL {X  -158.958, Y  +694.646, Z    +0.000, E1   -21.132, E3 +35157.458}
SPL {X  -159.960, Y  +679.609, Z    +0.000, E1    -6.021, E3 +35158.158}
SPL {X  -159.990, Y  +674.508, Z    +0.000, E1    -0.018, E3 +35158.217}
SPL {X  -159.990, Y  +672.787, Z    +0.000, E1    +4.022, E3 +35158.228}
SPL {X  -159.990, Y  +669.267, Z    +0.000, E1   +13.665, E3 +35158.299}
SPL {X  -159.990, Y  +665.069, Z    +0.000, E1   +25.376, E3 +35158.471}
SPL {X  -159.990, Y  +657.821, Z    +0.000, E1   +42.408, E3 +35158.973}
SPL {X  -159.990, Y  +645.368, Z    +0.000, E1   +59.257, E3 +35160.430}
SPL {X  -159.990, Y  +624.023, Z    +0.000, E1   +69.513, E3 +35164.554}
SPL {X  -159.990, Y  +543.075, Z    +0.000, E1   +75.590, E3 +35188.202}
SPL {X  -156.121, Y  +342.530, Z    +0.000, E1   +75.868, E3 +35274.849}
SPL {X  -153.865, Y  +333.657, Z    +0.000, E1   +75.438, E3 +35284.453}
ENDSPLINE

SPLINE
SPL {X  -159.103, Y  +360.678, Z    +0.000, E1   +72.233, E3 +35302.556}
ENDSPLINE

SPLINE
SPL {X  -154.371, Y  +335.471, Z    +0.000, E1   +73.016, E3 +35311.127}
SPL {X  -148.318, Y  +317.512, Z    +0.000, E1   +73.488, E3 +35317.448}
SPL {X  -141.230, Y  +302.327, Z    +0.000, E1   +73.933, E3 +35322.002}
SPL {X  -135.697, Y  +292.747, Z    +0.000, E1   +74.259, E3 +35324.360}
SPL {X  -132.590, Y  +287.964, Z    +0.000, E1   +73.910, E3 +35329.388}
SPL {X  -129.541, Y  +283.606, Z    +0.000, E1   +73.551, E3 +35334.029}
SPL {X  -126.457, Y  +279.493, Z    +0.000, E1   +73.175, E3 +35338.428}
SPL {X  -122.770, Y  +274.912, Z    +0.000, E1   +72.712, E3 +35343.283}
SPL {X  -119.156, Y  +270.736, Z    +0.000, E1   +72.213, E3 +35347.632}
SPL {X  -117.531, Y  +268.949, Z    +0.000, E1   +71.964, E3 +35349.448}
SPL {X   -74.907, Y  +236.129, Z    +0.000, E1   +61.720, E3 +35426.484}
SPL {X   -72.759, Y  +235.012, Z    +0.000, E1   +56.036, E3 +35598.161}
ENDSPLINE

SPLINE
SPL {X  -110.316, Y  +261.624, Z    +0.000, E1   +58.739, E3 +35670.234}
SPL {X  -136.558, Y  +294.141, Z    +0.000, E1   +54.887, E3 +35692.031}
SPL {X  -153.807, Y  +333.452, Z    +0.000, E1   +40.945, E3 +35702.428}
SPL {X  -158.168, Y  +353.421, Z    +0.000, E1   +27.296, E3 +35704.822}
SPL {X  -159.556, Y  +365.719, Z    +0.000, E1   +15.845, E3 +35705.623}
SPL {X  -159.982, Y  +375.924, Z    +0.000, E1    +4.476, E3 +35705.924}
SPL {X  -159.990, Y  +379.800, Z    +0.000, E1    -0.377, E3 +35705.953}
SPL {X  -159.990, Y  +383.422, Z    +0.000, E1   -10.730, E3 +35705.996}
SPL {X  -159.990, Y  +387.978, Z    +0.000, E1   -23.882, E3 +35706.148}
SPL {X  -159.990, Y  +394.494, Z    +0.000, E1   -40.961, E3 +35706.529}
SPL {X  -159.990, Y  +400.492, Z    +0.000, E1   -51.837, E3 +35707.053}
SPL {X  -159.990, Y  +409.662, Z    +0.000, E1   -61.705, E3 +35708.164}
SPL {X  -159.990, Y  +434.697, Z    +0.000, E1   -71.504, E3 +35713.184}
SPL {X  -159.990, Y  +521.523, Z    +0.000, E1   -76.035, E3 +35739.465}
SPL {X  -154.459, Y  +718.205, Z    +0.000, E1   -76.329, E3 +35821.260}
SPL {X  -151.356, Y  +728.349, Z    +0.000, E1   -76.056, E3 +35829.476}
SPL {X  -147.124, Y  +739.360, Z    +0.000, E1   -75.690, E3 +35839.072}
SPL {X  -142.861, Y  +748.524, Z    +0.000, E1   -75.261, E3 +35847.757}
SPL {X  -138.117, Y  +757.250, Z    +0.000, E1   -74.803, E3 +35856.360}
SPL {X  -133.491, Y  +764.686, Z    +0.000, E1   -74.276, E3 +35864.101}
SPL {X  -130.530, Y  +769.013, Z    +0.000, E1   -73.929, E3 +35868.683}
SPL {X  -127.734, Y  +772.837, Z    +0.000, E1   -73.601, E3 +35872.736}
SPL {X  -124.765, Y  +776.652, Z    +0.000, E1   -73.233, E3 +35876.770}
SPL {X  -121.376, Y  +780.734, Z    +0.000, E1   -72.804, E3 +35881.031}
SPL {X  -118.281, Y  +784.233, Z    +0.000, E1   -72.371, E3 +35884.600}
SPL {X   -72.391, Y  +819.176, Z    +0.000, E1   -59.867, E3 +35980.486}
ENDSPLINE

SPLINE
SPL {X  -116.241, Y  +786.431, Z    +0.000, E1   -57.120, E3 +36204.928}
SPL {X  -148.710, Y  +735.509, Z    +0.000, E1   -46.282, E3 +36230.660}
SPL {X  -157.559, Y  +704.285, Z    +0.000, E1   -29.037, E3 +36235.990}
SPL {X  -159.430, Y  +689.871, Z    +0.000, E1   -16.582, E3 +36237.140}
SPL {X  -159.960, Y  +679.609, Z    +0.000, E1    -6.021, E3 +36237.523}
SPL {X  -159.990, Y  +674.508, Z    +0.000, E1    -0.018, E3 +36237.582}
SPL {X  -159.990, Y  +672.787, Z    +0.000, E1    +4.022, E3 +36237.593}
SPL {X  -159.990, Y  +669.267, Z    +0.000, E1   +13.665, E3 +36237.664}
SPL {X  -159.990, Y  +665.069, Z    +0.000, E1   +25.376, E3 +36237.836}
SPL {X  -159.990, Y  +657.821, Z    +0.000, E1   +42.408, E3 +36238.338}
SPL {X  -159.990, Y  +645.368, Z    +0.000, E1   +59.257, E3 +36239.795}
SPL {X  -159.990, Y  +624.023, Z    +0.000, E1   +69.513, E3 +36243.919}
SPL {X  -159.990, Y  +543.075, Z    +0.000, E1   +75.590, E3 +36267.567}
SPL {X  -156.121, Y  +342.530, Z    +0.000, E1   +75.868, E3 +36354.214}
SPL {X  -153.865, Y  +333.657, Z    +0.000, E1   +75.438, E3 +36363.818}
ENDSPLINE

SPLINE
SPL {X  -159.644, Y  +366.989, Z    +0.000, E1   +72.058, E3 +36379.345}
ENDSPLINE

SPLINE
SPL {X  -156.933, Y  +346.374, Z    +0.000, E1   +72.645, E3 +36387.234}
SPL {X  -151.144, Y  +325.039, Z    +0.000, E1   +73.323, E3 +36393.914}
SPL {X  -145.016, Y  +309.920, Z    +0.000, E1   +73.647, E3 +36399.707}
SPL {X  -136.944, Y  +294.777, Z    +0.000, E1   +74.219, E3 +36403.009}
SPL {X  -132.590, Y  +287.964, Z    +0.000, E1   +73.910, E3 +36408.753}
SPL {X  -129.541, Y  +283.606, Z    +0.000, E1   +73.551, E3 +36413.394}
SPL {X  -125.403, Y  +278.147, Z    +0.000, E1   +73.063, E3 +36419.201}
SPL {X  -121.908, Y  +273.889, Z    +0.000, E1   +72.578, E3 +36423.747}
SPL {X  -118.941, Y  +270.496, Z    +0.000, E1   +72.188, E3 +36427.236}
SPL {X   -74.907, Y  +236.129, Z    +0.000, E1   +61.720, E3 +36505.849}
ENDSPLINE

SPLINE
SPL {X   -94.059, Y  +248.080, Z    +0.000, E1   +58.275, E3 +36727.542}
SPL {X  -136.558, Y  +294.141, Z    +0.000, E1   +54.887, E3 +36771.396}
SPL {X  -151.843, Y  +327.098, Z    +0.000, E1   +44.118, E3 +36780.756}
SPL {X  -157.484, Y  +349.293, Z    +0.000, E1   +30.654, E3 +36783.795}
SPL {X  -159.556, Y  +365.719, Z    +0.000, E1   +15.845, E3 +36784.988}
SPL {X  -159.982, Y  +375.924, Z    +0.000, E1    +4.476, E3 +36785.290}
SPL {X  -159.990, Y  +379.531, Z    +0.000, E1    -0.039, E3 +36785.317}
SPL {X  -159.990, Y  +382.420, Z    +0.000, E1    -7.600, E3 +36785.345}
SPL {X  -159.990, Y  +386.504, Z    +0.000, E1   -19.860, E3 +36785.450}
SPL {X  -159.990, Y  +392.530, Z    +0.000, E1   -36.133, E3 +36785.766}
SPL {X  -159.990, Y  +400.492, Z    +0.000, E1   -51.837, E3 +36786.418}
SPL {X  -159.990, Y  +409.662, Z    +0.000, E1   -61.705, E3 +36787.529}
SPL {X  -159.990, Y  +434.697, Z    +0.000, E1   -71.504, E3 +36792.549}
SPL {X  -159.990, Y  +521.523, Z    +0.000, E1   -76.035, E3 +36818.830}
SPL {X  -154.459, Y  +718.205, Z    +0.000, E1   -76.329, E3 +36900.625}
SPL {X  -151.356, Y  +728.349, Z    +0.000, E1   -76.056, E3 +36908.841}
SPL {X  -148.399, Y  +736.287, Z    +0.000, E1   -75.788, E3 +36915.719}
SPL {X  -144.005, Y  +746.209, Z    +0.000, E1   -75.396, E3 +36924.835}
SPL {X  -138.117, Y  +757.250, Z    +0.000, E1   -74.803, E3 +36935.726}
SPL {X  -133.491, Y  +764.686, Z    +0.000, E1   -74.276, E3 +36943.466}
SPL {X  -128.839, Y  +771.354, Z    +0.000, E1   -73.759, E3 +36950.485}
SPL {X  -123.568, Y  +778.125, Z    +0.000, E1   -73.105, E3 +36957.657}
SPL {X  -118.985, Y  +783.455, Z    +0.000, E1   -72.490, E3 +36963.164}
SPL {X   -72.391, Y  +819.176, Z    +0.000, E1   -59.867, E3 +37059.851}
ENDSPLINE

SPLINE
SPL {X   -92.809, Y  +806.820, Z    +0.000, E1   -56.994, E3 +37252.646}
SPL {X  -120.521, Y  +781.721, Z    +0.000, E1   -56.766, E3 +37288.745}
SPL {X  -143.482, Y  +747.279, Z    +0.000, E1   -50.227, E3 +37306.757}
SPL {X  -154.118, Y  +719.449, Z    +0.000, E1   -38.836, E3 +37313.337}
SPL {X  -158.281, Y  +699.823, Z    +0.000, E1   -25.469, E3 +37315.801}
SPL {X  -159.709, Y  +685.986, Z    +0.000, E1   -12.810, E3 +37316.687}
SPL {X  -159.990, Y  +674.648, Z    +0.000, E1    -0.349, E3 +37316.946}
SPL {X  -159.990, Y  +672.787, Z    +0.000, E1    +4.022, E3 +37316.959}
SPL {X  -159.990, Y  +669.267, Z    +0.000, E1   +13.665, E3 +37317.029}
SPL {X  -159.990, Y  +665.069, Z    +0.000, E1   +25.376, E3 +37317.201}
SPL {X  -159.990, Y  +657.821, Z    +0.000, E1   +42.408, E3 +37317.703}
SPL {X  -159.990, Y  +645.368, Z    +0.000, E1   +59.257, E3 +37319.160}
SPL {X  -159.990, Y  +624.023, Z    +0.000, E1   +69.513, E3 +37323.285}
SPL {X  -159.990, Y  +543.075, Z    +0.000, E1   +75.590, E3 +37346.933}
SPL {X  -156.121, Y  +342.530, Z    +0.000, E1   +75.868, E3 +37433.579}
SPL {X  -153.865, Y  +333.657, Z    +0.000, E1   +75.438, E3 +37443.183}
ENDSPLINE

SPLINE
SPL {X  -159.644, Y  +366.989, Z    +0.000, E1   +72.058, E3 +37458.710}
ENDSPLINE

SPLINE
SPL {X  -156.933, Y  +346.374, Z    +0.000, E1   +72.645, E3 +37466.599}
SPL {X  -151.144, Y  +325.039, Z    +0.000, E1   +73.323, E3 +37473.279}
SPL {X  -145.016, Y  +309.920, Z    +0.000, E1   +73.647, E3 +37479.072}
SPL {X  -136.944, Y  +294.777, Z    +0.000, E1   +74.219, E3 +37482.374}
SPL {X  -132.590, Y  +287.964, Z    +0.000, E1   +73.910, E3 +37488.118}
SPL {X  -129.541, Y  +283.606, Z    +0.000, E1   +73.551, E3 +37492.759}
SPL {X  -126.457, Y  +279.493, Z    +0.000, E1   +73.175, E3 +37497.158}
SPL {X  -122.770, Y  +274.912, Z    +0.000, E1   +72.712, E3 +37502.013}
SPL {X  -119.156, Y  +270.736, Z    +0.000, E1   +72.213, E3 +37506.363}
SPL {X  -117.531, Y  +268.949, Z    +0.000, E1   +71.964, E3 +37508.178}
SPL {X   -74.907, Y  +236.129, Z    +0.000, E1   +61.720, E3 +37585.214}
ENDSPLINE

SPLINE
SPL {X   -94.059, Y  +248.080, Z    +0.000, E1   +58.275, E3 +37806.907}
SPL {X  -130.769, Y  +285.325, Z    +0.000, E1   +56.495, E3 +37846.784}
SPL {X  -149.689, Y  +321.019, Z    +0.000, E1   +46.817, E3 +37858.868}
SPL {X  -157.484, Y  +349.293, Z    +0.000, E1   +30.654, E3 +37863.160}
SPL {X  -159.556, Y  +365.719, Z    +0.000, E1   +15.845, E3 +37864.353}
SPL {X  -159.982, Y  +375.924, Z    +0.000, E1    +4.476, E3 +37864.655}
SPL {X  -159.990, Y  +379.531, Z    +0.000, E1    -0.039, E3 +37864.682}
SPL {X  -159.990, Y  +382.420, Z    +0.000, E1    -7.600, E3 +37864.710}
SPL {X  -159.990, Y  +386.504, Z    +0.000, E1   -19.860, E3 +37864.815}
SPL {X  -159.990, Y  +392.530, Z    +0.000, E1   -36.133, E3 +37865.131}
SPL {X  -159.990, Y  +400.492, Z    +0.000, E1   -51.837, E3 +37865.783}
SPL {X  -159.990, Y  +409.662, Z    +0.000, E1   -61.705, E3 +37866.895}
SPL {X  -159.990, Y  +434.697, Z    +0.000, E1   -71.504, E3 +37871.915}
SPL {X  -159.990, Y  +521.523, Z    +0.000, E1   -76.035, E3 +37898.195}
SPL {X  -154.459, Y  +718.205, Z    +0.000, E1   -76.329, E3 +37979.990}
SPL {X  -151.356, Y  +728.349, Z    +0.000, E1   -76.056, E3 +37988.206}
SPL {X  -148.399, Y  +736.287, Z    +0.000, E1   -75.788, E3 +37995.085}
SPL {X  -144.005, Y  +746.209, Z    +0.000, E1   -75.396, E3 +38004.201}
SPL {X  -138.117, Y  +757.250, Z    +0.000, E1   -74.803, E3 +38015.091}
SPL {X  -133.491, Y  +764.686, Z    +0.000, E1   -74.276, E3 +38022.832}
SPL {X  -130.530, Y  +769.013, Z    +0.000, E1   -73.929, E3 +38027.413}
SPL {X  -127.734, Y  +772.837, Z    +0.000, E1   -73.601, E3 +38031.466}
SPL {X  -124.765, Y  +776.652, Z    +0.000, E1   -73.233, E3 +38035.500}
SPL {X  -121.376, Y  +780.734, Z    +0.000, E1   -72.804, E3 +38039.761}
SPL {X  -118.281, Y  +784.233, Z    +0.000, E1   -72.371, E3 +38043.330}
SPL {X   -72.391, Y  +819.176, Z    +0.000, E1   -59.867, E3 +38139.216}
ENDSPLINE

SPLINE
SPL {X  -116.241, Y  +786.431, Z    +0.000, E1   -57.120, E3 +38363.658}
SPL {X  -148.710, Y  +735.509, Z    +0.000, E1   -46.282, E3 +38389.391}
SPL {X  -157.559, Y  +704.285, Z    +0.000, E1   -29.037, E3 +38394.720}
SPL {X  -159.709, Y  +685.986, Z    +0.000, E1   -12.810, E3 +38396.052}
SPL {X  -159.990, Y  +674.648, Z    +0.000, E1    -0.349, E3 +38396.311}
SPL {X  -159.990, Y  +672.787, Z    +0.000, E1    +4.022, E3 +38396.324}
SPL {X  -159.990, Y  +669.267, Z    +0.000, E1   +13.665, E3 +38396.394}
SPL {X  -159.990, Y  +663.438, Z    +0.000, E1   +29.379, E3 +38396.665}
SPL {X  -159.990, Y  +655.264, Z    +0.000, E1   +47.291, E3 +38397.281}
SPL {X  -159.990, Y  +645.368, Z    +0.000, E1   +59.257, E3 +38398.525}
SPL {X  -159.990, Y  +624.023, Z    +0.000, E1   +69.513, E3 +38402.650}
SPL {X  -159.990, Y  +543.075, Z    +0.000, E1   +75.590, E3 +38426.298}
SPL {X  -156.121, Y  +342.530, Z    +0.000, E1   +75.868, E3 +38512.944}
SPL {X  -153.498, Y  +332.386, Z    +0.000, E1   +75.628, E3 +38520.948}
ENDSPLINE

SPLINE
SPL {X  -155.252, Y  +338.851, Z    +0.000, E1   +74.632, E3 +38528.327}
SPL {X  -159.103, Y  +360.678, Z    +0.000, E1   +72.233, E3 +38540.651}
ENDSPLINE

SPLINE
SPL {X  -154.371, Y  +335.471, Z    +0.000, E1   +73.016, E3 +38549.222}
SPL {X  -149.938, Y  +321.685, Z    +0.000, E1   +73.398, E3 +38553.917}
SPL {X  -145.016, Y  +309.920, Z    +0.000, E1   +73.647, E3 +38558.437}
SPL {X  -136.944, Y  +294.777, Z    +0.000, E1   +74.219, E3 +38561.739}
SPL {X  -132.590, Y  +287.964, Z    +0.000, E1   +73.910, E3 +38567.483}
SPL {X  -129.541, Y  +283.606, Z    +0.000, E1   +73.551, E3 +38572.124}
SPL {X  -125.403, Y  +278.147, Z    +0.000, E1   +73.063, E3 +38577.931}
SPL {X  -121.908, Y  +273.889, Z    +0.000, E1   +72.578, E3 +38582.478}
SPL {X  -119.156, Y  +270.736, Z    +0.000, E1   +72.213, E3 +38585.728}
SPL {X  -117.531, Y  +268.949, Z    +0.000, E1   +71.964, E3 +38587.543}
SPL {X   -74.907, Y  +236.129, Z    +0.000, E1   +61.720, E3 +38664.579}
ENDSPLINE

SPLINE
SPL {X   -94.059, Y  +248.080, Z    +0.000, E1   +58.275, E3 +38886.272}
SPL {X  -130.769, Y  +285.325, Z    +0.000, E1   +56.495, E3 +38926.149}
SPL {X  -149.689, Y  +321.019, Z    +0.000, E1   +46.817, E3 +38938.233}
SPL {X  -157.484, Y  +349.293, Z    +0.000, E1   +30.654, E3 +38942.526}
SPL {X  -159.556, Y  +365.719, Z    +0.000, E1   +15.845, E3 +38943.718}
SPL {X  -159.982, Y  +375.924, Z    +0.000, E1    +4.476, E3 +38944.020}
SPL {X  -159.990, Y  +379.531, Z    +0.000, E1    -0.039, E3 +38944.047}
SPL {X  -159.990, Y  +382.420, Z    +0.000, E1    -7.600, E3 +38944.075}
SPL {X  -159.990, Y  +386.504, Z    +0.000, E1   -19.860, E3 +38944.180}
SPL {X  -159.990, Y  +392.530, Z    +0.000, E1   -36.133, E3 +38944.496}
SPL {X  -159.990, Y  +400.492, Z    +0.000, E1   -51.837, E3 +38945.148}
SPL {X  -159.990, Y  +409.662, Z    +0.000, E1   -61.705, E3 +38946.260}
SPL {X  -159.990, Y  +434.697, Z    +0.000, E1   -71.504, E3 +38951.280}
SPL {X  -159.990, Y  +521.523, Z    +0.000, E1   -76.035, E3 +38977.560}
SPL {X  -154.459, Y  +718.205, Z    +0.000, E1   -76.329, E3 +39059.356}
SPL {X  -151.356, Y  +728.349, Z    +0.000, E1   -76.056, E3 +39067.571}
SPL {X  -148.399, Y  +736.287, Z    +0.000, E1   -75.788, E3 +39074.450}
SPL {X  -144.005, Y  +746.209, Z    +0.000, E1   -75.396, E3 +39083.566}
SPL {X  -138.117, Y  +757.250, Z    +0.000, E1   -74.803, E3 +39094.456}
SPL {X  -133.491, Y  +764.686, Z    +0.000, E1   -74.276, E3 +39102.197}
SPL {X  -128.839, Y  +771.354, Z    +0.000, E1   -73.759, E3 +39109.215}
SPL {X  -123.568, Y  +778.125, Z    +0.000, E1   -73.105, E3 +39116.387}
SPL {X  -118.985, Y  +783.455, Z    +0.000, E1   -72.490, E3 +39121.894}
SPL {X   -72.391, Y  +819.176, Z    +0.000, E1   -59.867, E3 +39218.581}
ENDSPLINE

SPLINE
SPL {X   -92.809, Y  +806.820, Z    +0.000, E1   -56.994, E3 +39411.376}
SPL {X  -120.521, Y  +781.721, Z    +0.000, E1   -56.766, E3 +39447.475}
SPL {X  -143.482, Y  +747.279, Z    +0.000, E1   -50.227, E3 +39465.488}
SPL {X  -154.118, Y  +719.449, Z    +0.000, E1   -38.836, E3 +39472.067}
SPL {X  -158.958, Y  +694.646, Z    +0.000, E1   -21.132, E3 +39474.918}
SPL {X  -159.960, Y  +679.609, Z    +0.000, E1    -6.021, E3 +39475.618}
SPL {X  -159.990, Y  +674.508, Z    +0.000, E1    -0.018, E3 +39475.677}
SPL {X  -159.990, Y  +672.787, Z    +0.000, E1    +4.022, E3 +39475.689}
SPL {X  -159.990, Y  +669.267, Z    +0.000, E1   +13.665, E3 +39475.759}
SPL {X  -159.990, Y  +663.438, Z    +0.000, E1   +29.379, E3 +39476.030}
SPL {X  -159.990, Y  +655.264, Z    +0.000, E1   +47.291, E3 +39476.647}
SPL {X  -159.990, Y  +645.368, Z    +0.000, E1   +59.257, E3 +39477.890}
SPL {X  -159.990, Y  +624.023, Z    +0.000, E1   +69.513, E3 +39482.015}
SPL {X  -159.990, Y  +543.075, Z    +0.000, E1   +75.590, E3 +39505.663}
SPL {X  -156.121, Y  +342.530, Z    +0.000, E1   +75.868, E3 +39592.309}
SPL {X  -153.498, Y  +332.386, Z    +0.000, E1   +75.628, E3 +39600.313}
ENDSPLINE

SPLINE
SPL {X  -155.252, Y  +338.851, Z    +0.000, E1   +74.632, E3 +39607.692}
SPL {X  -159.103, Y  +360.678, Z    +0.000, E1   +72.233, E3 +39620.017}
ENDSPLINE

SPLINE
SPL {X  -154.371, Y  +335.471, Z    +0.000, E1   +73.016, E3 +39628.587}
SPL {X  -149.938, Y  +321.685, Z    +0.000, E1   +73.398, E3 +39633.282}
SPL {X  -145.016, Y  +309.920, Z    +0.000, E1   +73.647, E3 +39637.803}
SPL {X  -139.138, Y  +298.522, Z    +0.000, E1   +74.138, E3 +39639.819}
SPL {X  -135.697, Y  +292.747, Z    +0.000, E1   +74.259, E3 +39641.820}
SPL {X  -132.590, Y  +287.964, Z    +0.000, E1   +73.910, E3 +39646.849}
SPL {X  -129.541, Y  +283.606, Z    +0.000, E1   +73.551, E3 +39651.489}
SPL {X  -126.457, Y  +279.493, Z    +0.000, E1   +73.175, E3 +39655.888}
SPL {X  -122.770, Y  +274.912, Z    +0.000, E1   +72.712, E3 +39660.743}
SPL {X  -118.941, Y  +270.496, Z    +0.000, E1   +72.188, E3 +39665.331}
SPL {X   -74.907, Y  +236.129, Z    +0.000, E1   +61.720, E3 +39743.944}
ENDSPLINE

SPLINE
SPL {X   -94.059, Y  +248.080, Z    +0.000, E1   +58.275, E3 +39965.637}
SPL {X  -136.558, Y  +294.141, Z    +0.000, E1   +54.887, E3 +40009.492}
SPL {X  -151.843, Y  +327.098, Z    +0.000, E1   +44.118, E3 +40018.851}
SPL {X  -157.484, Y  +349.293, Z    +0.000, E1   +30.654, E3 +40021.891}
SPL {X  -159.556, Y  +365.719, Z    +0.000, E1   +15.845, E3 +40023.083}
SPL {X  -159.982, Y  +375.924, Z    +0.000, E1    +4.476, E3 +40023.385}
SPL {X  -159.990, Y  +379.531, Z    +0.000, E1    -0.039, E3 +40023.412}
SPL {X  -159.990, Y  +382.420, Z    +0.000, E1    -7.600, E3 +40023.440}
SPL {X  -159.990, Y  +386.504, Z    +0.000, E1   -19.860, E3 +40023.546}
SPL {X  -159.990, Y  +392.530, Z    +0.000, E1   -36.133, E3 +40023.861}
SPL {X  -159.990, Y  +400.492, Z    +0.000, E1   -51.837, E3 +40024.514}
SPL {X  -159.990, Y  +409.662, Z    +0.000, E1   -61.705, E3 +40025.625}
SPL {X  -159.990, Y  +434.697, Z    +0.000, E1   -71.504, E3 +40030.645}
SPL {X  -159.990, Y  +521.523, Z    +0.000, E1   -76.035, E3 +40056.925}
SPL {X  -154.459, Y  +718.205, Z    +0.000, E1   -76.329, E3 +40138.721}
SPL {X  -151.356, Y  +728.349, Z    +0.000, E1   -76.056, E3 +40146.936}
SPL {X  -148.399, Y  +736.287, Z    +0.000, E1   -75.788, E3 +40153.815}
SPL {X  -144.005, Y  +746.209, Z    +0.000, E1   -75.396, E3 +40162.931}
SPL {X  -138.117, Y  +757.250, Z    +0.000, E1   -74.803, E3 +40173.821}
SPL {X  -133.491, Y  +764.686, Z    +0.000, E1   -74.276, E3 +40181.562}
SPL {X  -128.839, Y  +771.354, Z    +0.000, E1   -73.759, E3 +40188.580}
SPL {X  -123.568, Y  +778.125, Z    +0.000, E1   -73.105, E3 +40195.752}
SPL {X  -118.985, Y  +783.455, Z    +0.000, E1   -72.490, E3 +40201.260}
SPL {X   -72.391, Y  +819.176, Z    +0.000, E1   -59.867, E3 +40297.946}
ENDSPLINE

SPLINE
SPL {X   -92.809, Y  +806.820, Z    +0.000, E1   -56.994, E3 +40490.741}
SPL {X  -120.521, Y  +781.721, Z    +0.000, E1   -56.766, E3 +40526.840}
SPL {X  -148.710, Y  +735.509, Z    +0.000, E1   -46.282, E3 +40548.121}
SPL {X  -157.559, Y  +704.285, Z    +0.000, E1   -29.037, E3 +40553.450}
SPL {X  -159.430, Y  +689.871, Z    +0.000, E1   -16.582, E3 +40554.600}
SPL {X  -159.960, Y  +679.609, Z    +0.000, E1    -6.021, E3 +40554.983}
SPL {X  -159.990, Y  +674.508, Z    +0.000, E1    -0.018, E3 +40555.042}
SPL {X  -159.990, Y  +672.787, Z    +0.000, E1    +4.022, E3 +40555.054}
SPL {X  -159.990, Y  +669.267, Z    +0.000, E1   +13.665, E3 +40555.124}
SPL {X  -159.990, Y  +663.438, Z    +0.000, E1   +29.379, E3 +40555.395}
SPL {X  -159.990, Y  +655.264, Z    +0.000, E1   +47.291, E3 +40556.012}
SPL {X  -159.990, Y  +645.368, Z    +0.000, E1   +59.257, E3 +40557.255}
SPL {X  -159.990, Y  +624.023, Z    +0.000, E1   +69.513, E3 +40561.380}
SPL {X  -159.990, Y  +543.075, Z    +0.000, E1   +75.590, E3 +40585.028}
SPL {X  -156.121, Y  +342.530, Z    +0.000, E1   +75.868, E3 +40671.674}
SPL {X  -153.865, Y  +333.657, Z    +0.000, E1   +75.438, E3 +40681.278}
ENDSPLINE

SPLINE
SPL {X  -159.644, Y  +366.989, Z    +0.000, E1   +72.058, E3 +40696.805}
ENDSPLINE

SPLINE
SPL {X  -156.933, Y  +346.374, Z    +0.000, E1   +72.645, E3 +40704.694}
SPL {X  -151.144, Y  +325.039, Z    +0.000, E1   +73.323, E3 +40711.374}
SPL {X  -145.016, Y  +309.920, Z    +0.000, E1   +73.647, E3 +40717.168}
SPL {X  -136.944, Y  +294.777, Z    +0.000, E1   +74.219, E3 +40720.469}
SPL {X  -132.590, Y  +287.964, Z    +0.000, E1   +73.910, E3 +40726.214}
SPL {X  -129.541, Y  +283.606, Z    +0.000, E1   +73.551, E3 +40730.854}
SPL {X  -125.403, Y  +278.147, Z    +0.000, E1   +73.063, E3 +40736.661}
SPL {X  -121.908, Y  +273.889, Z    +0.000, E1   +72.578, E3 +40741.208}
SPL {X  -118.941, Y  +270.496, Z    +0.000, E1   +72.188, E3 +40744.696}
SPL {X   -74.907, Y  +236.129, Z    +0.000, E1   +61.720, E3 +40823.309}
ENDSPLINE

SPLINE
SPL {X   -94.059, Y  +248.080, Z    +0.000, E1   +58.275, E3 +41045.002}
SPL {X  -136.558, Y  +294.141, Z    +0.000, E1   +54.887, E3 +41088.857}
SPL {X  -151.843, Y  +327.098, Z    +0.000, E1   +44.118, E3 +41098.216}
SPL {X  -157.484, Y  +349.293, Z    +0.000, E1   +30.654, E3 +41101.256}
SPL {X  -159.556, Y  +365.719, Z    +0.000, E1   +15.845, E3 +41102.448}
SPL {X  -159.982, Y  +375.924, Z    +0.000, E1    +4.476, E3 +41102.750}
SPL {X  -159.990, Y  +379.531, Z    +0.000, E1    -0.039, E3 +41102.777}
SPL {X  -159.990, Y  +382.420, Z    +0.000, E1    -7.600, E3 +41102.805}
SPL {X  -159.990, Y  +386.504, Z    +0.000, E1   -19.860, E3 +41102.911}
SPL {X  -159.990, Y  +392.530, Z    +0.000, E1   -36.133, E3 +41103.226}
SPL {X  -159.990, Y  +400.492, Z    +0.000, E1   -51.837, E3 +41103.879}
SPL {X  -159.990, Y  +409.662, Z    +0.000, E1   -61.705, E3 +41104.990}
SPL {X  -159.990, Y  +434.697, Z    +0.000, E1   -71.504, E3 +41110.010}
SPL {X  -159.990, Y  +521.523, Z    +0.000, E1   -76.035, E3 +41136.290}
SPL {X  -154.459, Y  +718.205, Z    +0.000, E1   -76.329, E3 +41218.086}
SPL {X  -151.356, Y  +728.349, Z    +0.000, E1   -76.056, E3 +41226.301}
SPL {X  -148.399, Y  +736.287, Z    +0.000, E1   -75.788, E3 +41233.180}
SPL {X  -144.005, Y  +746.209, Z    +0.000, E1   -75.396, E3 +41242.296}
SPL {X  -138.117, Y  +757.250, Z    +0.000, E1   -74.803, E3 +41253.186}
SPL {X  -133.491, Y  +764.686, Z    +0.000, E1   -74.276, E3 +41260.927}
SPL {X  -128.839, Y  +771.354, Z    +0.000, E1   -73.759, E3 +41267.945}
SPL {X  -123.568, Y  +778.125, Z    +0.000, E1   -73.105, E3 +41275.117}
SPL {X  -118.985, Y  +783.455, Z    +0.000, E1   -72.490, E3 +41280.625}
SPL {X   -72.391, Y  +819.176, Z    +0.000, E1   -59.867, E3 +41377.311}
ENDSPLINE

SPLINE
SPL {X   -92.809, Y  +806.820, Z    +0.000, E1   -56.994, E3 +41570.106}
SPL {X  -120.521, Y  +781.721, Z    +0.000, E1   -56.766, E3 +41606.205}
SPL {X  -143.482, Y  +747.279, Z    +0.000, E1   -50.227, E3 +41624.218}
SPL {X  -154.118, Y  +719.449, Z    +0.000, E1   -38.836, E3 +41630.797}
SPL {X  -158.281, Y  +699.823, Z    +0.000, E1   -25.469, E3 +41633.262}
SPL {X  -159.709, Y  +685.986, Z    +0.000, E1   -12.810, E3 +41634.147}
SPL {X  -159.990, Y  +674.648, Z    +0.000, E1    -0.349, E3 +41634.406}
SPL {X  -159.990, Y  +672.787, Z    +0.000, E1    +4.022, E3 +41634.419}
SPL {X  -159.990, Y  +669.267, Z    +0.000, E1   +13.665, E3 +41634.489}
SPL {X  -159.990, Y  +663.438, Z    +0.000, E1   +29.379, E3 +41634.760}
SPL {X  -159.990, Y  +655.264, Z    +0.000, E1   +47.291, E3 +41635.377}
SPL {X  -159.990, Y  +645.368, Z    +0.000, E1   +59.257, E3 +41636.620}
SPL {X  -159.990, Y  +624.023, Z    +0.000, E1   +69.513, E3 +41640.745}
SPL {X  -159.990, Y  +543.075, Z    +0.000, E1   +75.590, E3 +41664.393}
SPL {X  -156.121, Y  +342.530, Z    +0.000, E1   +75.868, E3 +41751.039}
SPL {X  -153.865, Y  +333.657, Z    +0.000, E1   +75.438, E3 +41760.643}
ENDSPLINE

SPLINE
SPL {X  -159.644, Y  +366.989, Z    +0.000, E1   +72.058, E3 +41776.170}
ENDSPLINE

SPLINE
SPL {X  -156.933, Y  +346.374, Z    +0.000, E1   +72.645, E3 +41784.059}
SPL {X  -151.144, Y  +325.039, Z    +0.000, E1   +73.323, E3 +41790.739}
SPL {X  -145.016, Y  +309.920, Z    +0.000, E1   +73.647, E3 +41796.533}
SPL {X  -136.944, Y  +294.777, Z    +0.000, E1   +74.219, E3 +41799.834}
SPL {X  -132.590, Y  +287.964, Z    +0.000, E1   +73.910, E3 +41805.579}
SPL {X  -129.541, Y  +283.606, Z    +0.000, E1   +73.551, E3 +41810.219}
SPL {X  -125.403, Y  +278.147, Z    +0.000, E1   +73.063, E3 +41816.026}
SPL {X  -121.908, Y  +273.889, Z    +0.000, E1   +72.578, E3 +41820.573}
SPL {X  -118.941, Y  +270.496, Z    +0.000, E1   +72.188, E3 +41824.061}
SPL {X   -74.907, Y  +236.129, Z    +0.000, E1   +61.720, E3 +41902.674}
ENDSPLINE

SPLINE
SPL {X   -94.059, Y  +248.080, Z    +0.000, E1   +58.275, E3 +42124.367}
SPL {X  -136.558, Y  +294.141, Z    +0.000, E1   +54.887, E3 +42168.222}
SPL {X  -151.843, Y  +327.098, Z    +0.000, E1   +44.118, E3 +42177.581}
SPL {X  -157.484, Y  +349.293, Z    +0.000, E1   +30.654, E3 +42180.621}
SPL {X  -159.556, Y  +365.719, Z    +0.000, E1   +15.845, E3 +42181.813}
SPL {X  -159.982, Y  +375.924, Z    +0.000, E1    +4.476, E3 +42182.115}
SPL {X  -159.990, Y  +379.531, Z    +0.000, E1    -0.039, E3 +42182.142}
SPL {X  -159.990, Y  +382.420, Z    +0.000, E1    -7.600, E3 +42182.170}
SPL {X  -159.990, Y  +386.504, Z    +0.000, E1   -19.860, E3 +42182.276}
SPL {X  -159.990, Y  +392.530, Z    +0.000, E1   -36.133, E3 +42182.591}
SPL {X  -159.990, Y  +400.492, Z    +0.000, E1   -51.837, E3 +42183.244}
SPL {X  -159.990, Y  +409.662, Z    +0.000, E1   -61.705, E3 +42184.355}
SPL {X  -159.990, Y  +434.697, Z    +0.000, E1   -71.504, E3 +42189.375}
SPL {X  -159.990, Y  +521.523, Z    +0.000, E1   -76.035, E3 +42215.655}
SPL {X  -154.459, Y  +718.205, Z    +0.000, E1   -76.329, E3 +42297.451}
SPL {X  -151.356, Y  +728.349, Z    +0.000, E1   -76.056, E3 +42305.666}
SPL {X  -148.399, Y  +736.287, Z    +0.000, E1   -75.788, E3 +42312.545}
SPL {X  -144.005, Y  +746.209, Z    +0.000, E1   -75.396, E3 +42321.661}
SPL {X  -138.117, Y  +757.250, Z    +0.000, E1   -74.803, E3 +42332.551}
SPL {X  -133.491, Y  +764.686, Z    +0.000, E1   -74.276, E3 +42340.292}
SPL {X  -128.839, Y  +771.354, Z    +0.000, E1   -73.759, E3 +42347.311}
SPL {X  -123.568, Y  +778.125, Z    +0.000, E1   -73.105, E3 +42354.482}
SPL {X  -118.985, Y  +783.455, Z    +0.000, E1   -72.490, E3 +42359.990}
SPL {X   -72.391, Y  +819.176, Z    +0.000, E1   -59.867, E3 +42456.676}
ENDSPLINE

SPLINE
SPL {X   -92.809, Y  +806.820, Z    +0.000, E1   -56.994, E3 +42649.471}
SPL {X  -120.521, Y  +781.721, Z    +0.000, E1   -56.766, E3 +42685.570}
SPL {X  -143.482, Y  +747.279, Z    +0.000, E1   -50.227, E3 +42703.583}
SPL {X  -154.118, Y  +719.449, Z    +0.000, E1   -38.836, E3 +42710.162}
SPL {X  -158.958, Y  +694.646, Z    +0.000, E1   -21.132, E3 +42713.013}
SPL {X  -159.960, Y  +679.609, Z    +0.000, E1    -6.021, E3 +42713.714}
SPL {X  -159.990, Y  +674.508, Z    +0.000, E1    -0.018, E3 +42713.772}
SPL {X  -159.990, Y  +672.787, Z    +0.000, E1    +4.022, E3 +42713.784}
SPL {X  -159.990, Y  +669.267, Z    +0.000, E1   +13.665, E3 +42713.854}
SPL {X  -159.990, Y  +663.438, Z    +0.000, E1   +29.379, E3 +42714.125}
SPL {X  -159.990, Y  +655.264, Z    +0.000, E1   +47.291, E3 +42714.742}
SPL {X  -159.990, Y  +645.368, Z    +0.000, E1   +59.257, E3 +42715.985}
SPL {X  -159.990, Y  +624.023, Z    +0.000, E1   +69.513, E3 +42720.110}
SPL {X  -159.990, Y  +543.075, Z    +0.000, E1   +75.590, E3 +42743.758}
SPL {X  -156.121, Y  +342.530, Z    +0.000, E1   +75.868, E3 +42830.404}
SPL {X  -153.498, Y  +332.386, Z    +0.000, E1   +75.628, E3 +42838.409}
ENDSPLINE

SPLINE
SPL {X  -155.252, Y  +338.851, Z    +0.000, E1   +74.632, E3 +42845.787}
SPL {X  -159.103, Y  +360.678, Z    +0.000, E1   +72.233, E3 +42858.112}
ENDSPLINE

SPLINE
SPL {X  -154.371, Y  +335.471, Z    +0.000, E1   +73.016, E3 +42866.683}
SPL {X  -149.938, Y  +321.685, Z    +0.000, E1   +73.398, E3 +42871.377}
SPL {X  -145.016, Y  +309.920, Z    +0.000, E1   +73.647, E3 +42875.898}
SPL {X  -139.138, Y  +298.522, Z    +0.000, E1   +74.138, E3 +42877.914}
SPL {X  -135.697, Y  +292.747, Z    +0.000, E1   +74.259, E3 +42879.916}
SPL {X  -132.590, Y  +287.964, Z    +0.000, E1   +73.910, E3 +42884.944}
SPL {X  -129.541, Y  +283.606, Z    +0.000, E1   +73.551, E3 +42889.584}
SPL {X  -126.457, Y  +279.493, Z    +0.000, E1   +73.175, E3 +42893.983}
SPL {X  -122.770, Y  +274.912, Z    +0.000, E1   +72.712, E3 +42898.839}
SPL {X  -118.941, Y  +270.496, Z    +0.000, E1   +72.188, E3 +42903.426}
SPL {X   -74.907, Y  +236.129, Z    +0.000, E1   +61.720, E3 +42982.039}
ENDSPLINE

SPLINE
SPL {X   -94.059, Y  +248.080, Z    +0.000, E1   +58.275, E3 +43203.732}
SPL {X  -136.558, Y  +294.141, Z    +0.000, E1   +54.887, E3 +43247.587}
SPL {X  -151.843, Y  +327.098, Z    +0.000, E1   +44.118, E3 +43256.946}
SPL {X  -157.484, Y  +349.293, Z    +0.000, E1   +30.654, E3 +43259.986}
SPL {X  -159.556, Y  +365.719, Z    +0.000, E1   +15.845, E3 +43261.178}
SPL {X  -159.982, Y  +375.924, Z    +0.000, E1    +4.476, E3 +43261.480}
SPL {X  -159.990, Y  +379.531, Z    +0.000, E1    -0.039, E3 +43261.507}
SPL {X  -159.990, Y  +382.420, Z    +0.000, E1    -7.600, E3 +43261.535}
SPL {X  -159.990, Y  +386.504, Z    +0.000, E1   -19.860, E3 +43261.641}
SPL {X  -159.990, Y  +392.530, Z    +0.000, E1   -36.133, E3 +43261.956}
SPL {X  -159.990, Y  +400.492, Z    +0.000, E1   -51.837, E3 +43262.609}
SPL {X  -159.990, Y  +409.662, Z    +0.000, E1   -61.705, E3 +43263.720}
SPL {X  -159.990, Y  +434.697, Z    +0.000, E1   -71.504, E3 +43268.740}
SPL {X  -159.990, Y  +521.523, Z    +0.000, E1   -76.035, E3 +43295.021}
SPL {X  -154.459, Y  +718.205, Z    +0.000, E1   -76.329, E3 +43376.816}
SPL {X  -151.356, Y  +728.349, Z    +0.000, E1   -76.056, E3 +43385.031}
SPL {X  -148.399, Y  +736.287, Z    +0.000, E1   -75.788, E3 +43391.910}
SPL {X  -144.005, Y  +746.209, Z    +0.000, E1   -75.396, E3 +43401.026}
SPL {X  -138.117, Y  +757.250, Z    +0.000, E1   -74.803, E3 +43411.916}
SPL {X  -133.491, Y  +764.686, Z    +0.000, E1   -74.276, E3 +43419.657}
SPL {X  -130.530, Y  +769.013, Z    +0.000, E1   -73.929, E3 +43424.239}
SPL {X  -127.734, Y  +772.837, Z    +0.000, E1   -73.601, E3 +43428.291}
SPL {X  -124.765, Y  +776.652, Z    +0.000, E1   -73.233, E3 +43432.326}
SPL {X  -121.376, Y  +780.734, Z    +0.000, E1   -72.804, E3 +43436.587}
SPL {X  -118.281, Y  +784.233, Z    +0.000, E1   -72.371, E3 +43440.155}
SPL {X   -72.391, Y  +819.176, Z    +0.000, E1   -59.867, E3 +43536.041}
ENDSPLINE

SPLINE
SPL {X   -92.809, Y  +806.820, Z    +0.000, E1   -56.994, E3 +43728.836}
SPL {X  -120.521, Y  +781.721, Z    +0.000, E1   -56.766, E3 +43764.935}
SPL {X  -143.482, Y  +747.279, Z    +0.000, E1   -50.227, E3 +43782.948}
SPL {X  -154.118, Y  +719.449, Z    +0.000, E1   -38.836, E3 +43789.527}
SPL {X  -158.958, Y  +694.646, Z    +0.000, E1   -21.132, E3 +43792.379}
SPL {X  -159.960, Y  +679.609, Z    +0.000, E1    -6.021, E3 +43793.079}
SPL {X  -159.990, Y  +674.508, Z    +0.000, E1    -0.018, E3 +43793.137}
SPL {X  -159.990, Y  +672.787, Z    +0.000, E1    +4.022, E3 +43793.149}
SPL {X  -159.990, Y  +669.267, Z    +0.000, E1   +13.665, E3 +43793.219}
SPL {X  -159.990, Y  +665.069, Z    +0.000, E1   +25.376, E3 +43793.391}
SPL {X  -159.990, Y  +657.821, Z    +0.000, E1   +42.408, E3 +43793.893}
SPL {X  -159.990, Y  +645.368, Z    +0.000, E1   +59.257, E3 +43795.350}
SPL {X  -159.990, Y  +624.023, Z    +0.000, E1   +69.513, E3 +43799.475}
SPL {X  -159.990, Y  +543.075, Z    +0.000, E1   +75.590, E3 +43823.123}
SPL {X  -156.121, Y  +342.530, Z    +0.000, E1   +75.868, E3 +43909.769}
SPL {X  -153.865, Y  +333.657, Z    +0.000, E1   +75.438, E3 +43919.373}
ENDSPLINE

SPLINE
SPL {X  -159.103, Y  +360.678, Z    +0.000, E1   +72.233, E3 +43937.477}
ENDSPLINE

SPLINE
SPL {X  -154.371, Y  +335.471, Z    +0.000, E1   +73.016, E3 +43946.048}
SPL {X  -148.318, Y  +317.512, Z    +0.000, E1   +73.488, E3 +43952.369}
SPL {X  -141.230, Y  +302.327, Z    +0.000, E1   +73.933, E3 +43956.922}
SPL {X  -135.697, Y  +292.747, Z    +0.000, E1   +74.259, E3 +43959.281}
SPL {X  -132.590, Y  +287.964, Z    +0.000, E1   +73.910, E3 +43964.309}
SPL {X  -129.541, Y  +283.606, Z    +0.000, E1   +73.551, E3 +43968.949}
SPL {X  -126.457, Y  +279.493, Z    +0.000, E1   +73.175, E3 +43973.348}
SPL {X  -122.770, Y  +274.912, Z    +0.000, E1   +72.712, E3 +43978.204}
SPL {X  -119.156, Y  +270.736, Z    +0.000, E1   +72.213, E3 +43982.553}
SPL {X  -117.531, Y  +268.949, Z    +0.000, E1   +71.964, E3 +43984.369}
SPL {X   -74.907, Y  +236.129, Z    +0.000, E1   +61.720, E3 +44061.404}
SPL {X   -72.759, Y  +235.012, Z    +0.000, E1   +56.036, E3 +44233.082}
ENDSPLINE

SPLINE
SPL {X  -110.316, Y  +261.624, Z    +0.000, E1   +58.739, E3 +44305.155}
SPL {X  -136.558, Y  +294.141, Z    +0.000, E1   +54.887, E3 +44326.952}
SPL {X  -153.807, Y  +333.452, Z    +0.000, E1   +40.945, E3 +44337.349}
SPL {X  -158.168, Y  +353.421, Z    +0.000, E1   +27.296, E3 +44339.742}
SPL {X  -159.556, Y  +365.719, Z    +0.000, E1   +15.845, E3 +44340.543}
SPL {X  -159.982, Y  +375.924, Z    +0.000, E1    +4.476, E3 +44340.845}
SPL {X  -159.990, Y  +379.800, Z    +0.000, E1    -0.377, E3 +44340.874}
SPL {X  -159.990, Y  +383.422, Z    +0.000, E1   -10.730, E3 +44340.916}
SPL {X  -159.990, Y  +387.978, Z    +0.000, E1   -23.882, E3 +44341.069}
SPL {X  -159.990, Y  +394.494, Z    +0.000, E1   -40.961, E3 +44341.450}
SPL {X  -159.990, Y  +400.492, Z    +0.000, E1   -51.837, E3 +44341.974}
SPL {X  -159.990, Y  +409.662, Z    +0.000, E1   -61.705, E3 +44343.085}
SPL {X  -159.990, Y  +434.697, Z    +0.000, E1   -71.504, E3 +44348.105}
SPL {X  -159.990, Y  +521.523, Z    +0.000, E1   -76.035, E3 +44374.386}
SPL {X  -154.459, Y  +718.205, Z    +0.000, E1   -76.329, E3 +44456.181}
SPL {X  -151.356, Y  +728.349, Z    +0.000, E1   -76.056, E3 +44464.397}
SPL {X  -147.124, Y  +739.360, Z    +0.000, E1   -75.690, E3 +44473.993}
SPL {X  -142.861, Y  +748.524, Z    +0.000, E1   -75.261, E3 +44482.678}
SPL {X  -139.796, Y  +754.307, Z    +0.000, E1   -74.951, E3 +44488.366}
SPL {X  -136.850, Y  +759.378, Z    +0.000, E1   -74.643, E3 +44493.510}
SPL {X  -133.491, Y  +764.686, Z    +0.000, E1   -74.276, E3 +44499.022}
SPL {X  -128.839, Y  +771.354, Z    +0.000, E1   -73.759, E3 +44506.041}
SPL {X  -123.568, Y  +778.125, Z    +0.000, E1   -73.105, E3 +44513.212}
SPL {X  -118.985, Y  +783.455, Z    +0.000, E1   -72.490, E3 +44518.720}
SPL {X   -72.391, Y  +819.176, Z    +0.000, E1   -59.867, E3 +44615.406}
ENDSPLINE

SPLINE
SPL {X   -92.809, Y  +806.820, Z    +0.000, E1   -56.994, E3 +44808.201}
SPL {X  -120.521, Y  +781.721, Z    +0.000, E1   -56.766, E3 +44844.300}
SPL {X  -148.710, Y  +735.509, Z    +0.000, E1   -46.282, E3 +44865.581}
SPL {X  -157.559, Y  +704.285, Z    +0.000, E1   -29.037, E3 +44870.910}
SPL {X  -159.430, Y  +689.871, Z    +0.000, E1   -16.582, E3 +44872.061}
SPL {X  -159.960, Y  +679.609, Z    +0.000, E1    -6.021, E3 +44872.444}
SPL {X  -159.990, Y  +674.508, Z    +0.000, E1    -0.018, E3 +44872.502}
SPL {X  -159.990, Y  +672.787, Z    +0.000, E1    +4.022, E3 +44872.514}
SPL {X  -159.990, Y  +669.267, Z    +0.000, E1   +13.665, E3 +44872.584}
SPL {X  -159.990, Y  +663.438, Z    +0.000, E1   +29.379, E3 +44872.855}
SPL {X  -159.990, Y  +655.264, Z    +0.000, E1   +47.291, E3 +44873.472}
SPL {X  -159.990, Y  +645.368, Z    +0.000, E1   +59.257, E3 +44874.715}
SPL {X  -159.990, Y  +624.023, Z    +0.000, E1   +69.513, E3 +44878.840}
SPL {X  -159.990, Y  +543.075, Z    +0.000, E1   +75.590, E3 +44902.488}
SPL {X  -156.121, Y  +342.530, Z    +0.000, E1   +75.868, E3 +44989.134}
SPL {X  -153.865, Y  +333.657, Z    +0.000, E1   +75.438, E3 +44998.738}
ENDSPLINE

SPLINE
SPL {X  -159.644, Y  +366.989, Z    +0.000, E1   +72.058, E3 +45014.265}
ENDSPLINE

SPLINE
SPL {X  -156.933, Y  +346.374, Z    +0.000, E1   +72.645, E3 +45022.154}
SPL {X  -151.144, Y  +325.039, Z    +0.000, E1   +73.323, E3 +45028.834}
SPL {X  -146.668, Y  +313.584, Z    +0.000, E1   +73.560, E3 +45033.316}
SPL {X  -141.230, Y  +302.327, Z    +0.000, E1   +73.933, E3 +45036.287}
SPL {X  -135.697, Y  +292.747, Z    +0.000, E1   +74.259, E3 +45038.646}
SPL {X  -132.590, Y  +287.964, Z    +0.000, E1   +73.910, E3 +45043.674}
SPL {X  -129.541, Y  +283.606, Z    +0.000, E1   +73.551, E3 +45048.315}
SPL {X  -125.403, Y  +278.147, Z    +0.000, E1   +73.063, E3 +45054.122}
SPL {X  -121.908, Y  +273.889, Z    +0.000, E1   +72.578, E3 +45058.668}
SPL {X  -119.156, Y  +270.736, Z    +0.000, E1   +72.213, E3 +45061.918}
SPL {X  -117.531, Y  +268.949, Z    +0.000, E1   +71.964, E3 +45063.734}
SPL {X   -74.907, Y  +236.129, Z    +0.000, E1   +61.720, E3 +45140.770}
ENDSPLINE

SPLINE
SPL {X   -94.059, Y  +248.080, Z    +0.000, E1   +58.275, E3 +45362.462}
SPL {X  -130.769, Y  +285.325, Z    +0.000, E1   +56.495, E3 +45402.339}
SPL {X  -149.689, Y  +321.019, Z    +0.000, E1   +46.817, E3 +45414.424}
SPL {X  -157.484, Y  +349.293, Z    +0.000, E1   +30.654, E3 +45418.716}
SPL {X  -159.556, Y  +365.719, Z    +0.000, E1   +15.845, E3 +45419.909}
SPL {X  -159.982, Y  +375.924, Z    +0.000, E1    +4.476, E3 +45420.210}
SPL {X  -159.990, Y  +379.531, Z    +0.000, E1    -0.039, E3 +45420.237}
SPL {X  -159.990, Y  +382.420, Z    +0.000, E1    -7.600, E3 +45420.266}
SPL {X  -159.990, Y  +386.504, Z    +0.000, E1   -19.860, E3 +45420.371}
SPL {X  -159.990, Y  +392.530, Z    +0.000, E1   -36.133, E3 +45420.686}
SPL {X  -159.990, Y  +400.492, Z    +0.000, E1   -51.837, E3 +45421.339}
SPL {X  -159.990, Y  +409.662, Z    +0.000, E1   -61.705, E3 +45422.450}
SPL {X  -159.990, Y  +434.697, Z    +0.000, E1   -71.504, E3 +45427.470}
SPL {X  -159.990, Y  +521.523, Z    +0.000, E1   -76.035, E3 +45453.751}
SPL {X  -154.459, Y  +718.205, Z    +0.000, E1   -76.329, E3 +45535.546}
SPL {X  -151.356, Y  +728.349, Z    +0.000, E1   -76.056, E3 +45543.762}
SPL {X  -147.124, Y  +739.360, Z    +0.000, E1   -75.690, E3 +45553.358}
SPL {X  -142.861, Y  +748.524, Z    +0.000, E1   -75.261, E3 +45562.043}
SPL {X  -139.796, Y  +754.307, Z    +0.000, E1   -74.951, E3 +45567.731}
SPL {X  -136.850, Y  +759.378, Z    +0.000, E1   -74.643, E3 +45572.875}
SPL {X  -133.491, Y  +764.686, Z    +0.000, E1   -74.276, E3 +45578.387}
SPL {X  -130.530, Y  +769.013, Z    +0.000, E1   -73.929, E3 +45582.969}
SPL {X  -127.734, Y  +772.837, Z    +0.000, E1   -73.601, E3 +45587.021}
SPL {X  -123.568, Y  +778.125, Z    +0.000, E1   -73.105, E3 +45592.578}
SPL {X  -118.985, Y  +783.455, Z    +0.000, E1   -72.490, E3 +45598.085}
SPL {X   -72.391, Y  +819.176, Z    +0.000, E1   -59.867, E3 +45694.771}
ENDSPLINE

SPLINE
SPL {X   -92.809, Y  +806.820, Z    +0.000, E1   -56.994, E3 +45887.566}
SPL {X  -120.521, Y  +781.721, Z    +0.000, E1   -56.766, E3 +45923.665}
SPL {X  -148.710, Y  +735.509, Z    +0.000, E1   -46.282, E3 +45944.946}
SPL {X  -157.559, Y  +704.285, Z    +0.000, E1   -29.037, E3 +45950.276}
SPL {X  -159.709, Y  +685.986, Z    +0.000, E1   -12.810, E3 +45951.607}
SPL {X  -159.990, Y  +674.648, Z    +0.000, E1    -0.349, E3 +45951.867}
SPL {X  -159.990, Y  +672.787, Z    +0.000, E1    +4.022, E3 +45951.879}
SPL {X  -159.990, Y  +669.267, Z    +0.000, E1   +13.665, E3 +45951.949}
SPL {X  -159.990, Y  +665.069, Z    +0.000, E1   +25.376, E3 +45952.121}
SPL {X  -159.990, Y  +657.821, Z    +0.000, E1   +42.408, E3 +45952.624}
SPL {X  -159.990, Y  +645.368, Z    +0.000, E1   +59.257, E3 +45954.080}
SPL {X  -159.990, Y  +624.023, Z    +0.000, E1   +69.513, E3 +45958.205}
SPL {X  -159.990, Y  +543.075, Z    +0.000, E1   +75.590, E3 +45981.853}
SPL {X  -156.121, Y  +342.530, Z    +0.000, E1   +75.868, E3 +46068.499}
SPL {X  -153.865, Y  +333.657, Z    +0.000, E1   +75.438, E3 +46078.103}
ENDSPLINE

SPLINE
SPL {X  -159.644, Y  +366.989, Z    +0.000, E1   +72.058, E3 +46093.630}
ENDSPLINE

SPLINE
SPL {X  -156.933, Y  +346.374, Z    +0.000, E1   +72.645, E3 +46101.520}
SPL {X  -151.144, Y  +325.039, Z    +0.000, E1   +73.323, E3 +46108.199}
SPL {X  -145.016, Y  +309.920, Z    +0.000, E1   +73.647, E3 +46113.993}
SPL {X  -136.944, Y  +294.777, Z    +0.000, E1   +74.219, E3 +46117.295}
SPL {X  -132.590, Y  +287.964, Z    +0.000, E1   +73.910, E3 +46123.039}
SPL {X  -129.541, Y  +283.606, Z    +0.000, E1   +73.551, E3 +46127.680}
SPL {X  -126.457, Y  +279.493, Z    +0.000, E1   +73.175, E3 +46132.079}
SPL {X  -122.770, Y  +274.912, Z    +0.000, E1   +72.712, E3 +46136.934}
SPL {X  -119.156, Y  +270.736, Z    +0.000, E1   +72.213, E3 +46141.283}
SPL {X  -117.531, Y  +268.949, Z    +0.000, E1   +71.964, E3 +46143.099}
SPL {X   -74.907, Y  +236.129, Z    +0.000, E1   +61.720, E3 +46220.135}
SPL {X   -72.759, Y  +235.012, Z    +0.000, E1   +56.036, E3 +46391.812}
ENDSPLINE

SPLINE
SPL {X  -110.316, Y  +261.624, Z    +0.000, E1   +58.739, E3 +46463.885}
SPL {X  -136.558, Y  +294.141, Z    +0.000, E1   +54.887, E3 +46485.682}
SPL {X  -153.807, Y  +333.452, Z    +0.000, E1   +40.945, E3 +46496.079}
SPL {X  -158.168, Y  +353.421, Z    +0.000, E1   +27.296, E3 +46498.472}
SPL {X  -159.556, Y  +365.719, Z    +0.000, E1   +15.845, E3 +46499.274}
SPL {X  -159.982, Y  +375.924, Z    +0.000, E1    +4.476, E3 +46499.575}
SPL {X  -159.990, Y  +379.800, Z    +0.000, E1    -0.377, E3 +46499.604}
SPL {X  -159.990, Y  +383.422, Z    +0.000, E1   -10.730, E3 +46499.647}
SPL {X  -159.990, Y  +387.978, Z    +0.000, E1   -23.882, E3 +46499.799}
SPL {X  -159.990, Y  +394.494, Z    +0.000, E1   -40.961, E3 +46500.180}
SPL {X  -159.990, Y  +400.492, Z    +0.000, E1   -51.837, E3 +46500.704}
SPL {X  -159.990, Y  +409.662, Z    +0.000, E1   -61.705, E3 +46501.815}
SPL {X  -159.990, Y  +434.697, Z    +0.000, E1   -71.504, E3 +46506.835}
SPL {X  -159.990, Y  +521.523, Z    +0.000, E1   -76.035, E3 +46533.116}
SPL {X  -154.459, Y  +718.205, Z    +0.000, E1   -76.329, E3 +46614.911}
SPL {X  -151.356, Y  +728.349, Z    +0.000, E1   -76.056, E3 +46623.127}
SPL {X  -148.399, Y  +736.287, Z    +0.000, E1   -75.788, E3 +46630.005}
SPL {X  -144.005, Y  +746.209, Z    +0.000, E1   -75.396, E3 +46639.121}
SPL {X  -138.117, Y  +757.250, Z    +0.000, E1   -74.803, E3 +46650.011}
SPL {X  -133.491, Y  +764.686, Z    +0.000, E1   -74.276, E3 +46657.752}
SPL {X  -128.839, Y  +771.354, Z    +0.000, E1   -73.759, E3 +46664.771}
SPL {X  -124.765, Y  +776.652, Z    +0.000, E1   -73.233, E3 +46670.421}
SPL {X  -121.376, Y  +780.734, Z    +0.000, E1   -72.804, E3 +46674.682}
SPL {X  -118.281, Y  +784.233, Z    +0.000, E1   -72.371, E3 +46678.251}
SPL {X   -72.391, Y  +819.176, Z    +0.000, E1   -59.867, E3 +46774.136}
ENDSPLINE

SPLINE
SPL {X  -116.241, Y  +786.431, Z    +0.000, E1   -57.120, E3 +46998.579}
SPL {X  -143.482, Y  +747.279, Z    +0.000, E1   -50.227, E3 +47021.043}
SPL {X  -154.118, Y  +719.449, Z    +0.000, E1   -38.836, E3 +47027.623}
SPL {X  -158.958, Y  +694.646, Z    +0.000, E1   -21.132, E3 +47030.474}
SPL {X  -159.960, Y  +679.609, Z    +0.000, E1    -6.021, E3 +47031.174}
SPL {X  -159.990, Y  +674.508, Z    +0.000, E1    -0.018, E3 +47031.233}
SPL {X  -159.990, Y  +672.787, Z    +0.000, E1    +4.022, E3 +47031.244}
SPL {X  -159.990, Y  +669.267, Z    +0.000, E1   +13.665, E3 +47031.315}
SPL {X  -159.990, Y  +665.069, Z    +0.000, E1   +25.376, E3 +47031.486}
SPL {X  -159.990, Y  +657.821, Z    +0.000, E1   +42.408, E3 +47031.989}
SPL {X  -159.990, Y  +645.368, Z    +0.000, E1   +59.257, E3 +47033.445}
SPL {X  -159.990, Y  +624.023, Z    +0.000, E1   +69.513, E3 +47037.570}
SPL {X  -159.990, Y  +543.075, Z    +0.000, E1   +75.590, E3 +47061.218}
SPL {X  -156.121, Y  +342.530, Z    +0.000, E1   +75.868, E3 +47147.864}
SPL {X  -153.865, Y  +333.657, Z    +0.000, E1   +75.438, E3 +47157.468}
ENDSPLINE

SPLINE
SPL {X  -159.644, Y  +366.989, Z    +0.000, E1   +72.058, E3 +47172.995}
ENDSPLINE

SPLINE
SPL {X  -156.933, Y  +346.374, Z    +0.000, E1   +72.645, E3 +47180.885}
SPL {X  -151.144, Y  +325.039, Z    +0.000, E1   +73.323, E3 +47187.564}
SPL {X  -145.016, Y  +309.920, Z    +0.000, E1   +73.647, E3 +47193.358}
SPL {X  -136.944, Y  +294.777, Z    +0.000, E1   +74.219, E3 +47196.660}
SPL {X  -132.590, Y  +287.964, Z    +0.000, E1   +73.910, E3 +47202.404}
SPL {X  -129.541, Y  +283.606, Z    +0.000, E1   +73.551, E3 +47207.045}
SPL {X  -126.457, Y  +279.493, Z    +0.000, E1   +73.175, E3 +47211.444}
SPL {X  -122.770, Y  +274.912, Z    +0.000, E1   +72.712, E3 +47216.299}
SPL {X  -119.156, Y  +270.736, Z    +0.000, E1   +72.213, E3 +47220.648}
SPL {X  -117.531, Y  +268.949, Z    +0.000, E1   +71.964, E3 +47222.464}
SPL {X   -74.907, Y  +236.129, Z    +0.000, E1   +61.720, E3 +47299.500}
ENDSPLINE

SPLINE
SPL {X   -94.059, Y  +248.080, Z    +0.000, E1   +58.275, E3 +47521.193}
SPL {X  -130.769, Y  +285.325, Z    +0.000, E1   +56.495, E3 +47561.070}
SPL {X  -149.689, Y  +321.019, Z    +0.000, E1   +46.817, E3 +47573.154}
SPL {X  -155.950, Y  +341.772, Z    +0.000, E1   +35.915, E3 +47576.652}
SPL {X  -158.168, Y  +353.421, Z    +0.000, E1   +27.296, E3 +47577.838}
SPL {X  -159.556, Y  +365.719, Z    +0.000, E1   +15.845, E3 +47578.639}
SPL {X  -159.982, Y  +375.924, Z    +0.000, E1    +4.476, E3 +47578.940}
SPL {X  -159.990, Y  +379.800, Z    +0.000, E1    -0.377, E3 +47578.969}
SPL {X  -159.990, Y  +383.422, Z    +0.000, E1   -10.730, E3 +47579.012}
SPL {X  -159.990, Y  +387.978, Z    +0.000, E1   -23.882, E3 +47579.164}
SPL {X  -159.990, Y  +394.494, Z    +0.000, E1   -40.961, E3 +47579.545}
SPL {X  -159.990, Y  +400.492, Z    +0.000, E1   -51.837, E3 +47580.069}
SPL {X  -159.990, Y  +409.662, Z    +0.000, E1   -61.705, E3 +47581.180}
SPL {X  -159.990, Y  +434.697, Z    +0.000, E1   -71.504, E3 +47586.200}
SPL {X  -159.990, Y  +521.523, Z    +0.000, E1   -76.035, E3 +47612.481}
SPL {X  -154.459, Y  +718.205, Z    +0.000, E1   -76.329, E3 +47694.276}
SPL {X  -151.356, Y  +728.349, Z    +0.000, E1   -76.056, E3 +47702.492}
SPL {X  -147.124, Y  +739.360, Z    +0.000, E1   -75.690, E3 +47712.088}
SPL {X  -142.861, Y  +748.524, Z    +0.000, E1   -75.261, E3 +47720.773}
SPL {X  -139.796, Y  +754.307, Z    +0.000, E1   -74.951, E3 +47726.461}
SPL {X  -136.850, Y  +759.378, Z    +0.000, E1   -74.643, E3 +47731.606}
SPL {X  -133.491, Y  +764.686, Z    +0.000, E1   -74.276, E3 +47737.117}
SPL {X  -128.839, Y  +771.354, Z    +0.000, E1   -73.759, E3 +47744.136}
SPL {X  -124.765, Y  +776.652, Z    +0.000, E1   -73.233, E3 +47749.786}
SPL {X  -121.376, Y  +780.734, Z    +0.000, E1   -72.804, E3 +47754.047}
SPL {X  -118.281, Y  +784.233, Z    +0.000, E1   -72.371, E3 +47757.616}
SPL {X   -72.391, Y  +819.176, Z    +0.000, E1   -59.867, E3 +47853.501}
ENDSPLINE

SPLINE
SPL {X  -116.241, Y  +786.431, Z    +0.000, E1   -57.120, E3 +48077.944}
SPL {X  -143.482, Y  +747.279, Z    +0.000, E1   -50.227, E3 +48100.408}
SPL {X  -154.118, Y  +719.449, Z    +0.000, E1   -38.836, E3 +48106.988}
SPL {X  -158.958, Y  +694.646, Z    +0.000, E1   -21.132, E3 +48109.839}
SPL {X  -159.960, Y  +679.609, Z    +0.000, E1    -6.021, E3 +48110.539}
SPL {X  -159.990, Y  +674.508, Z    +0.000, E1    -0.018, E3 +48110.598}
SPL {X  -159.990, Y  +672.787, Z    +0.000, E1    +4.022, E3 +48110.609}
SPL {X  -159.990, Y  +669.267, Z    +0.000, E1   +13.665, E3 +48110.680}
SPL {X  -159.990, Y  +665.069, Z    +0.000, E1   +25.376, E3 +48110.851}
SPL {X  -159.990, Y  +657.821, Z    +0.000, E1   +42.408, E3 +48111.354}
SPL {X  -159.990, Y  +645.368, Z    +0.000, E1   +59.257, E3 +48112.811}
SPL {X  -159.990, Y  +624.023, Z    +0.000, E1   +69.513, E3 +48116.935}
SPL {X  -159.990, Y  +543.075, Z    +0.000, E1   +75.590, E3 +48140.583}
SPL {X  -156.121, Y  +342.530, Z    +0.000, E1   +75.868, E3 +48227.230}
SPL {X  -153.865, Y  +333.657, Z    +0.000, E1   +75.438, E3 +48236.834}
ENDSPLINE

SPLINE
SPL {X  -159.103, Y  +360.678, Z    +0.000, E1   +72.233, E3 +48254.937}
ENDSPLINE

SPLINE
SPL {X  -154.371, Y  +335.471, Z    +0.000, E1   +73.016, E3 +48263.508}
SPL {X  -148.318, Y  +317.512, Z    +0.000, E1   +73.488, E3 +48269.829}
SPL {X  -141.230, Y  +302.327, Z    +0.000, E1   +73.933, E3 +48274.383}
SPL {X  -135.697, Y  +292.747, Z    +0.000, E1   +74.259, E3 +48276.741}
SPL {X  -132.590, Y  +287.964, Z    +0.000, E1   +73.910, E3 +48281.769}
SPL {X  -129.541, Y  +283.606, Z    +0.000, E1   +73.551, E3 +48286.410}
SPL {X  -126.457, Y  +279.493, Z    +0.000, E1   +73.175, E3 +48290.809}
SPL {X  -122.770, Y  +274.912, Z    +0.000, E1   +72.712, E3 +48295.664}
SPL {X  -118.941, Y  +270.496, Z    +0.000, E1   +72.188, E3 +48300.252}
SPL {X   -74.907, Y  +236.129, Z    +0.000, E1   +61.720, E3 +48378.865}
SPL {X   -72.759, Y  +235.012, Z    +0.000, E1   +56.036, E3 +48550.542}
ENDSPLINE

SPLINE
SPL {X  -123.257, Y  +275.497, Z    +0.000, E1   +57.800, E3 +48634.418}
SPL {X  -149.689, Y  +321.019, Z    +0.000, E1   +46.817, E3 +48652.519}
SPL {X  -157.484, Y  +349.293, Z    +0.000, E1   +30.654, E3 +48656.811}
SPL {X  -159.556, Y  +365.719, Z    +0.000, E1   +15.845, E3 +48658.004}
SPL {X  -159.982, Y  +375.924, Z    +0.000, E1    +4.476, E3 +48658.305}
SPL {X  -159.990, Y  +379.531, Z    +0.000, E1    -0.039, E3 +48658.332}
SPL {X  -159.990, Y  +382.420, Z    +0.000, E1    -7.600, E3 +48658.361}
SPL {X  -159.990, Y  +387.978, Z    +0.000, E1   -23.882, E3 +48658.529}
SPL {X  -159.990, Y  +396.850, Z    +0.000, E1   -45.459, E3 +48659.116}
SPL {X  -159.990, Y  +409.662, Z    +0.000, E1   -61.705, E3 +48660.545}
SPL {X  -159.990, Y  +434.697, Z    +0.000, E1   -71.504, E3 +48665.565}
SPL {X  -159.990, Y  +521.523, Z    +0.000, E1   -76.035, E3 +48691.846}
SPL {X  -154.459, Y  +718.205, Z    +0.000, E1   -76.329, E3 +48773.641}
SPL {X  -151.356, Y  +728.349, Z    +0.000, E1   -76.056, E3 +48781.857}
SPL {X  -148.399, Y  +736.287, Z    +0.000, E1   -75.788, E3 +48788.735}
SPL {X  -144.005, Y  +746.209, Z    +0.000, E1   -75.396, E3 +48797.851}
SPL {X  -138.117, Y  +757.250, Z    +0.000, E1   -74.803, E3 +48808.741}
SPL {X  -133.491, Y  +764.686, Z    +0.000, E1   -74.276, E3 +48816.482}
SPL {X  -128.839, Y  +771.354, Z    +0.000, E1   -73.759, E3 +48823.501}
SPL {X  -124.765, Y  +776.652, Z    +0.000, E1   -73.233, E3 +48829.151}
SPL {X  -121.376, Y  +780.734, Z    +0.000, E1   -72.804, E3 +48833.412}
SPL {X  -118.281, Y  +784.233, Z    +0.000, E1   -72.371, E3 +48836.981}
SPL {X   -72.391, Y  +819.176, Z    +0.000, E1   -59.867, E3 +48932.867}
ENDSPLINE

SPLINE
SPL {X  -116.241, Y  +786.431, Z    +0.000, E1   -57.120, E3 +49157.309}
SPL {X  -148.710, Y  +735.509, Z    +0.000, E1   -46.282, E3 +49183.041}
SPL {X  -157.559, Y  +704.285, Z    +0.000, E1   -29.037, E3 +49188.371}
SPL {X  -159.709, Y  +685.986, Z    +0.000, E1   -12.810, E3 +49189.702}
SPL {X  -159.990, Y  +674.648, Z    +0.000, E1    -0.349, E3 +49189.962}
SPL {X  -159.990, Y  +672.787, Z    +0.000, E1    +4.022, E3 +49189.974}
SPL {X  -159.990, Y  +669.267, Z    +0.000, E1   +13.665, E3 +49190.045}
SPL {X  -159.990, Y  +663.438, Z    +0.000, E1   +29.379, E3 +49190.315}
SPL {X  -159.990, Y  +655.264, Z    +0.000, E1   +47.291, E3 +49190.932}
SPL {X  -159.990, Y  +645.368, Z    +0.000, E1   +59.257, E3 +49192.176}
SPL {X  -159.990, Y  +624.023, Z    +0.000, E1   +69.513, E3 +49196.300}
SPL {X  -159.990, Y  +543.075, Z    +0.000, E1   +75.590, E3 +49219.948}
SPL {X  -156.121, Y  +342.530, Z    +0.000, E1   +75.868, E3 +49306.595}
SPL {X  -153.498, Y  +332.386, Z    +0.000, E1   +75.628, E3 +49314.599}
ENDSPLINE

SPLINE
SPL {X  -155.252, Y  +338.851, Z    +0.000, E1   +74.632, E3 +49321.977}
SPL {X  -159.103, Y  +360.678, Z    +0.000, E1   +72.233, E3 +49334.302}
ENDSPLINE

SPLINE
SPL {X  -154.371, Y  +335.471, Z    +0.000, E1   +73.016, E3 +49342.873}
SPL {X  -149.938, Y  +321.685, Z    +0.000, E1   +73.398, E3 +49347.567}
SPL {X  -145.016, Y  +309.920, Z    +0.000, E1   +73.647, E3 +49352.088}
SPL {X  -136.944, Y  +294.777, Z    +0.000, E1   +74.219, E3 +49355.390}
SPL {X  -132.590, Y  +287.964, Z    +0.000, E1   +73.910, E3 +49361.134}
SPL {X  -129.541, Y  +283.606, Z    +0.000, E1   +73.551, E3 +49365.775}
SPL {X  -125.403, Y  +278.147, Z    +0.000, E1   +73.063, E3 +49371.582}
SPL {X  -121.908, Y  +273.889, Z    +0.000, E1   +72.578, E3 +49376.128}
SPL {X  -119.156, Y  +270.736, Z    +0.000, E1   +72.213, E3 +49379.378}
SPL {X  -117.531, Y  +268.949, Z    +0.000, E1   +71.964, E3 +49381.194}
SPL {X   -74.907, Y  +236.129, Z    +0.000, E1   +61.720, E3 +49458.230}
ENDSPLINE

SPLINE
SPL {X   -94.059, Y  +248.080, Z    +0.000, E1   +58.275, E3 +49679.923}
SPL {X  -130.769, Y  +285.325, Z    +0.000, E1   +56.495, E3 +49719.800}
SPL {X  -149.689, Y  +321.019, Z    +0.000, E1   +46.817, E3 +49731.884}
SPL {X  -157.484, Y  +349.293, Z    +0.000, E1   +30.654, E3 +49736.176}
SPL {X  -159.556, Y  +365.719, Z    +0.000, E1   +15.845, E3 +49737.369}
SPL {X  -159.982, Y  +375.924, Z    +0.000, E1    +4.476, E3 +49737.670}
SPL {X  -159.990, Y  +379.531, Z    +0.000, E1    -0.039, E3 +49737.697}
SPL {X  -159.990, Y  +382.420, Z    +0.000, E1    -7.600, E3 +49737.726}
SPL {X  -159.990, Y  +386.504, Z    +0.000, E1   -19.860, E3 +49737.831}
SPL {X  -159.990, Y  +392.530, Z    +0.000, E1   -36.133, E3 +49738.146}
SPL {X  -159.990, Y  +400.492, Z    +0.000, E1   -51.837, E3 +49738.799}
SPL {X  -159.990, Y  +409.662, Z    +0.000, E1   -61.705, E3 +49739.910}
SPL {X  -159.990, Y  +434.697, Z    +0.000, E1   -71.504, E3 +49744.930}
SPL {X  -159.990, Y  +521.523, Z    +0.000, E1   -76.035, E3 +49771.211}
SPL {X  -154.459, Y  +718.205, Z    +0.000, E1   -76.329, E3 +49853.006}
SPL {X  -151.356, Y  +728.349, Z    +0.000, E1   -76.056, E3 +49861.222}
SPL {X  -148.399, Y  +736.287, Z    +0.000, E1   -75.788, E3 +49868.100}
SPL {X  -144.005, Y  +746.209, Z    +0.000, E1   -75.396, E3 +49877.216}
SPL {X  -138.117, Y  +757.250, Z    +0.000, E1   -74.803, E3 +49888.106}
SPL {X  -133.491, Y  +764.686, Z    +0.000, E1   -74.276, E3 +49895.847}
SPL {X  -128.839, Y  +771.354, Z    +0.000, E1   -73.759, E3 +49902.866}
SPL {X  -123.568, Y  +778.125, Z    +0.000, E1   -73.105, E3 +49910.038}
SPL {X  -118.985, Y  +783.455, Z    +0.000, E1   -72.490, E3 +49915.545}
SPL {X   -72.391, Y  +819.176, Z    +0.000, E1   -59.867, E3 +50012.232}
ENDSPLINE

SPLINE
SPL {X   -92.809, Y  +806.820, Z    +0.000, E1   -56.994, E3 +50205.027}
SPL {X  -120.521, Y  +781.721, Z    +0.000, E1   -56.766, E3 +50241.126}
SPL {X  -143.482, Y  +747.279, Z    +0.000, E1   -50.227, E3 +50259.138}
SPL {X  -154.118, Y  +719.449, Z    +0.000, E1   -38.836, E3 +50265.718}
SPL {X  -158.958, Y  +694.646, Z    +0.000, E1   -21.132, E3 +50268.569}
SPL {X  -159.960, Y  +679.609, Z    +0.000, E1    -6.021, E3 +50269.269}
SPL {X  -159.990, Y  +674.508, Z    +0.000, E1    -0.018, E3 +50269.328}
SPL {X  -159.990, Y  +672.787, Z    +0.000, E1    +4.022, E3 +50269.340}
SPL {X  -159.990, Y  +669.267, Z    +0.000, E1   +13.665, E3 +50269.410}
SPL {X  -159.990, Y  +663.438, Z    +0.000, E1   +29.379, E3 +50269.680}
SPL {X  -159.990, Y  +655.264, Z    +0.000, E1   +47.291, E3 +50270.297}
SPL {X  -159.990, Y  +645.368, Z    +0.000, E1   +59.257, E3 +50271.541}
SPL {X  -159.990, Y  +624.023, Z    +0.000, E1   +69.513, E3 +50275.665}
SPL {X  -159.990, Y  +543.075, Z    +0.000, E1   +75.590, E3 +50299.313}
SPL {X  -156.121, Y  +342.530, Z    +0.000, E1   +75.868, E3 +50385.960}
SPL {X  -153.498, Y  +332.386, Z    +0.000, E1   +75.628, E3 +50393.964}
ENDSPLINE

SPLINE
SPL {X  -155.252, Y  +338.851, Z    +0.000, E1   +74.632, E3 +50401.342}
SPL {X  -159.103, Y  +360.678, Z    +0.000, E1   +72.233, E3 +50413.667}
ENDSPLINE

SPLINE
SPL {X  -154.371, Y  +335.471, Z    +0.000, E1   +73.016, E3 +50422.238}
SPL {X  -149.938, Y  +321.685, Z    +0.000, E1   +73.398, E3 +50426.933}
SPL {X  -145.016, Y  +309.920, Z    +0.000, E1   +73.647, E3 +50431.453}
SPL {X  -139.138, Y  +298.522, Z    +0.000, E1   +74.138, E3 +50433.469}
SPL {X  -135.697, Y  +292.747, Z    +0.000, E1   +74.259, E3 +50435.471}
SPL {X  -132.590, Y  +287.964, Z    +0.000, E1   +73.910, E3 +50440.499}
SPL {X  -129.541, Y  +283.606, Z    +0.000, E1   +73.551, E3 +50445.140}
SPL {X  -126.457, Y  +279.493, Z    +0.000, E1   +73.175, E3 +50449.539}
SPL {X  -122.770, Y  +274.912, Z    +0.000, E1   +72.712, E3 +50454.394}
SPL {X  -118.941, Y  +270.496, Z    +0.000, E1   +72.188, E3 +50458.982}
SPL {X   -74.907, Y  +236.129, Z    +0.000, E1   +61.720, E3 +50537.595}
ENDSPLINE

SPLINE
SPL {X   -94.059, Y  +248.080, Z    +0.000, E1   +58.275, E3 +50759.288}
SPL {X  -136.558, Y  +294.141, Z    +0.000, E1   +54.887, E3 +50803.142}
SPL {X  -151.843, Y  +327.098, Z    +0.000, E1   +44.118, E3 +50812.502}
SPL {X  -157.484, Y  +349.293, Z    +0.000, E1   +30.654, E3 +50815.541}
SPL {X  -159.556, Y  +365.719, Z    +0.000, E1   +15.845, E3 +50816.734}
SPL {X  -159.982, Y  +375.924, Z    +0.000, E1    +4.476, E3 +50817.036}
SPL {X  -159.990, Y  +379.531, Z    +0.000, E1    -0.039, E3 +50817.063}
SPL {X  -159.990, Y  +382.420, Z    +0.000, E1    -7.600, E3 +50817.091}
SPL {X  -159.990, Y  +386.504, Z    +0.000, E1   -19.860, E3 +50817.196}
SPL {X  -159.990, Y  +392.530, Z    +0.000, E1   -36.133, E3 +50817.512}
SPL {X  -159.990, Y  +400.492, Z    +0.000, E1   -51.837, E3 +50818.164}
SPL {X  -159.990, Y  +409.662, Z    +0.000, E1   -61.705, E3 +50819.276}
SPL {X  -159.990, Y  +434.697, Z    +0.000, E1   -71.504, E3 +50824.295}
SPL {X  -159.990, Y  +521.523, Z    +0.000, E1   -76.035, E3 +50850.576}
SPL {X  -154.459, Y  +718.205, Z    +0.000, E1   -76.329, E3 +50932.371}
SPL {X  -151.356, Y  +728.349, Z    +0.000, E1   -76.056, E3 +50940.587}
SPL {X  -148.399, Y  +736.287, Z    +0.000, E1   -75.788, E3 +50947.466}
SPL {X  -144.005, Y  +746.209, Z    +0.000, E1   -75.396, E3 +50956.581}
SPL {X  -138.117, Y  +757.250, Z    +0.000, E1   -74.803, E3 +50967.472}
SPL {X  -133.491, Y  +764.686, Z    +0.000, E1   -74.276, E3 +50975.212}
SPL {X  -130.530, Y  +769.013, Z    +0.000, E1   -73.929, E3 +50979.794}
SPL {X  -127.734, Y  +772.837, Z    +0.000, E1   -73.601, E3 +50983.847}
SPL {X  -124.765, Y  +776.652, Z    +0.000, E1   -73.233, E3 +50987.881}
SPL {X  -121.376, Y  +780.734, Z    +0.000, E1   -72.804, E3 +50992.142}
SPL {X  -118.281, Y  +784.233, Z    +0.000, E1   -72.371, E3 +50995.711}
SPL {X   -72.391, Y  +819.176, Z    +0.000, E1   -59.867, E3 +51091.597}
ENDSPLINE

SPLINE
SPL {X   -92.809, Y  +806.820, Z    +0.000, E1   -56.994, E3 +51284.392}
SPL {X  -120.521, Y  +781.721, Z    +0.000, E1   -56.766, E3 +51320.491}
SPL {X  -143.482, Y  +747.279, Z    +0.000, E1   -50.227, E3 +51338.504}
SPL {X  -154.118, Y  +719.449, Z    +0.000, E1   -38.836, E3 +51345.083}
SPL {X  -158.958, Y  +694.646, Z    +0.000, E1   -21.132, E3 +51347.934}
SPL {X  -159.960, Y  +679.609, Z    +0.000, E1    -6.021, E3 +51348.634}
SPL {X  -159.990, Y  +674.508, Z    +0.000, E1    -0.018, E3 +51348.693}
SPL {X  -159.990, Y  +672.787, Z    +0.000, E1    +4.022, E3 +51348.705}
SPL {X  -159.990, Y  +669.267, Z    +0.000, E1   +13.665, E3 +51348.775}
SPL {X  -159.990, Y  +665.069, Z    +0.000, E1   +25.376, E3 +51348.947}
SPL {X  -159.990, Y  +657.821, Z    +0.000, E1   +42.408, E3 +51349.449}
SPL {X  -159.990, Y  +645.368, Z    +0.000, E1   +59.257, E3 +51350.906}
SPL {X  -159.990, Y  +624.023, Z    +0.000, E1   +69.513, E3 +51355.031}
SPL {X  -159.990, Y  +543.075, Z    +0.000, E1   +75.590, E3 +51378.679}
SPL {X  -156.121, Y  +342.530, Z    +0.000, E1   +75.868, E3 +51465.325}
SPL {X  -153.865, Y  +333.657, Z    +0.000, E1   +75.438, E3 +51474.929}
ENDSPLINE

SPLINE
SPL {X  -159.103, Y  +360.678, Z    +0.000, E1   +72.233, E3 +51493.032}
ENDSPLINE

SPLINE
SPL {X  -154.371, Y  +335.471, Z    +0.000, E1   +73.016, E3 +51501.603}
SPL {X  -148.318, Y  +317.512, Z    +0.000, E1   +73.488, E3 +51507.924}
SPL {X  -141.230, Y  +302.327, Z    +0.000, E1   +73.933, E3 +51512.478}
SPL {X  -135.697, Y  +292.747, Z    +0.000, E1   +74.259, E3 +51514.836}
SPL {X  -132.590, Y  +287.964, Z    +0.000, E1   +73.910, E3 +51519.864}
SPL {X  -129.541, Y  +283.606, Z    +0.000, E1   +73.551, E3 +51524.505}
SPL {X  -126.457, Y  +279.493, Z    +0.000, E1   +73.175, E3 +51528.904}
SPL {X  -122.770, Y  +274.912, Z    +0.000, E1   +72.712, E3 +51533.759}
SPL {X  -119.156, Y  +270.736, Z    +0.000, E1   +72.213, E3 +51538.109}
SPL {X  -117.531, Y  +268.949, Z    +0.000, E1   +71.964, E3 +51539.924}
SPL {X   -74.907, Y  +236.129, Z    +0.000, E1   +61.720, E3 +51616.960}
SPL {X   -72.759, Y  +235.012, Z    +0.000, E1   +56.036, E3 +51788.638}
ENDSPLINE

SPLINE
SPL {X  -110.316, Y  +261.624, Z    +0.000, E1   +58.739, E3 +51860.710}
SPL {X  -136.558, Y  +294.141, Z    +0.000, E1   +54.887, E3 +51882.507}
SPL {X  -153.807, Y  +333.452, Z    +0.000, E1   +40.945, E3 +51892.904}
SPL {X  -158.168, Y  +353.421, Z    +0.000, E1   +27.296, E3 +51895.298}
SPL {X  -159.556, Y  +365.719, Z    +0.000, E1   +15.845, E3 +51896.099}
SPL {X  -159.982, Y  +375.924, Z    +0.000, E1    +4.476, E3 +51896.401}
SPL {X  -159.990, Y  +379.800, Z    +0.000, E1    -0.377, E3 +51896.429}
SPL {X  -159.990, Y  +383.422, Z    +0.000, E1   -10.730, E3 +51896.472}
SPL {X  -159.990, Y  +387.978, Z    +0.000, E1   -23.882, E3 +51896.624}
SPL {X  -159.990, Y  +394.494, Z    +0.000, E1   -40.961, E3 +51897.005}
SPL {X  -159.990, Y  +400.492, Z    +0.000, E1   -51.837, E3 +51897.529}
SPL {X  -159.990, Y  +409.662, Z    +0.000, E1   -61.705, E3 +51898.641}
SPL {X  -159.990, Y  +434.697, Z    +0.000, E1   -71.504, E3 +51903.661}
SPL {X  -159.990, Y  +521.523, Z    +0.000, E1   -76.035, E3 +51929.941}
SPL {X  -154.459, Y  +718.205, Z    +0.000, E1   -76.329, E3 +52011.736}
SPL {X  -151.356, Y  +728.349, Z    +0.000, E1   -76.056, E3 +52019.952}
SPL {X  -147.124, Y  +739.360, Z    +0.000, E1   -75.690, E3 +52029.548}
SPL {X  -142.861, Y  +748.524, Z    +0.000, E1   -75.261, E3 +52038.233}
SPL {X  -138.117, Y  +757.250, Z    +0.000, E1   -74.803, E3 +52046.837}
SPL {X  -133.491, Y  +764.686, Z    +0.000, E1   -74.276, E3 +52054.578}
SPL {X  -130.530, Y  +769.013, Z    +0.000, E1   -73.929, E3 +52059.159}
SPL {X  -127.734, Y  +772.837, Z    +0.000, E1   -73.601, E3 +52063.212}
SPL {X  -124.765, Y  +776.652, Z    +0.000, E1   -73.233, E3 +52067.246}
SPL {X  -121.376, Y  +780.734, Z    +0.000, E1   -72.804, E3 +52071.508}
SPL {X  -118.281, Y  +784.233, Z    +0.000, E1   -72.371, E3 +52075.076}
SPL {X   -72.391, Y  +819.176, Z    +0.000, E1   -59.867, E3 +52170.962}
ENDSPLINE

SPLINE
SPL {X  -116.241, Y  +786.431, Z    +0.000, E1   -57.120, E3 +52395.404}
SPL {X  -148.710, Y  +735.509, Z    +0.000, E1   -46.282, E3 +52421.137}
SPL {X  -157.559, Y  +704.285, Z    +0.000, E1   -29.037, E3 +52426.466}
SPL {X  -159.430, Y  +689.871, Z    +0.000, E1   -16.582, E3 +52427.616}
SPL {X  -159.960, Y  +679.609, Z    +0.000, E1    -6.021, E3 +52427.999}
SPL {X  -159.990, Y  +674.508, Z    +0.000, E1    -0.018, E3 +52428.058}
SPL {X  -159.990, Y  +672.787, Z    +0.000, E1    +4.022, E3 +52428.070}
SPL {X  -159.990, Y  +669.267, Z    +0.000, E1   +13.665, E3 +52428.140}
SPL {X  -159.990, Y  +663.438, Z    +0.000, E1   +29.379, E3 +52428.411}
SPL {X  -159.990, Y  +655.264, Z    +0.000, E1   +47.291, E3 +52429.027}
SPL {X  -159.990, Y  +645.368, Z    +0.000, E1   +59.257, E3 +52430.271}
SPL {X  -159.990, Y  +624.023, Z    +0.000, E1   +69.513, E3 +52434.396}
SPL {X  -159.990, Y  +543.075, Z    +0.000, E1   +75.590, E3 +52458.044}
SPL {X  -156.121, Y  +342.530, Z    +0.000, E1   +75.868, E3 +52544.690}
SPL {X  -153.498, Y  +332.386, Z    +0.000, E1   +75.628, E3 +52552.694}
ENDSPLINE

SPLINE
SPL {X  -155.252, Y  +338.851, Z    +0.000, E1   +74.632, E3 +52560.073}
SPL {X  -159.103, Y  +360.678, Z    +0.000, E1   +72.233, E3 +52572.398}
ENDSPLINE

SPLINE
SPL {X  -154.371, Y  +335.471, Z    +0.000, E1   +73.016, E3 +52580.968}
SPL {X  -149.938, Y  +321.685, Z    +0.000, E1   +73.398, E3 +52585.663}
SPL {X  -145.016, Y  +309.920, Z    +0.000, E1   +73.647, E3 +52590.183}
SPL {X  -139.138, Y  +298.522, Z    +0.000, E1   +74.138, E3 +52592.200}
SPL {X  -135.697, Y  +292.747, Z    +0.000, E1   +74.259, E3 +52594.201}
SPL {X  -132.590, Y  +287.964, Z    +0.000, E1   +73.910, E3 +52599.229}
SPL {X  -129.541, Y  +283.606, Z    +0.000, E1   +73.551, E3 +52603.870}
SPL {X  -126.457, Y  +279.493, Z    +0.000, E1   +73.175, E3 +52608.269}
SPL {X  -122.770, Y  +274.912, Z    +0.000, E1   +72.712, E3 +52613.124}
SPL {X  -119.156, Y  +270.736, Z    +0.000, E1   +72.213, E3 +52617.474}
SPL {X  -117.531, Y  +268.949, Z    +0.000, E1   +71.964, E3 +52619.289}
SPL {X   -74.907, Y  +236.129, Z    +0.000, E1   +61.720, E3 +52696.325}
ENDSPLINE

SPLINE
SPL {X   -94.059, Y  +248.080, Z    +0.000, E1   +58.275, E3 +52918.018}
SPL {X  -130.769, Y  +285.325, Z    +0.000, E1   +56.495, E3 +52957.895}
SPL {X  -149.689, Y  +321.019, Z    +0.000, E1   +46.817, E3 +52969.979}
SPL {X  -157.484, Y  +349.293, Z    +0.000, E1   +30.654, E3 +52974.272}
SPL {X  -159.556, Y  +365.719, Z    +0.000, E1   +15.845, E3 +52975.464}
SPL {X  -159.982, Y  +375.924, Z    +0.000, E1    +4.476, E3 +52975.766}
SPL {X  -159.990, Y  +379.531, Z    +0.000, E1    -0.039, E3 +52975.793}
SPL {X  -159.990, Y  +382.420, Z    +0.000, E1    -7.600, E3 +52975.821}
SPL {X  -159.990, Y  +386.504, Z    +0.000, E1   -19.860, E3 +52975.927}
SPL {X  -159.990, Y  +392.530, Z    +0.000, E1   -36.133, E3 +52976.242}
SPL {X  -159.990, Y  +400.492, Z    +0.000, E1   -51.837, E3 +52976.895}
SPL {X  -159.990, Y  +409.662, Z    +0.000, E1   -61.705, E3 +52978.006}
SPL {X  -159.990, Y  +434.697, Z    +0.000, E1   -71.504, E3 +52983.026}
SPL {X  -159.990, Y  +521.523, Z    +0.000, E1   -76.035, E3 +53009.306}
SPL {X  -154.459, Y  +718.205, Z    +0.000, E1   -76.329, E3 +53091.102}
SPL {X  -151.356, Y  +728.349, Z    +0.000, E1   -76.056, E3 +53099.317}
SPL {X  -148.399, Y  +736.287, Z    +0.000, E1   -75.788, E3 +53106.196}
SPL {X  -144.005, Y  +746.209, Z    +0.000, E1   -75.396, E3 +53115.312}
SPL {X  -138.117, Y  +757.250, Z    +0.000, E1   -74.803, E3 +53126.202}
SPL {X  -133.491, Y  +764.686, Z    +0.000, E1   -74.276, E3 +53133.943}
SPL {X  -128.839, Y  +771.354, Z    +0.000, E1   -73.759, E3 +53140.961}
SPL {X  -123.568, Y  +778.125, Z    +0.000, E1   -73.105, E3 +53148.133}
SPL {X  -118.985, Y  +783.455, Z    +0.000, E1   -72.490, E3 +53153.640}
SPL {X   -72.391, Y  +819.176, Z    +0.000, E1   -59.867, E3 +53250.327}
ENDSPLINE

SPLINE
SPL {X   -92.809, Y  +806.820, Z    +0.000, E1   -56.994, E3 +53443.122}
SPL {X  -120.521, Y  +781.721, Z    +0.000, E1   -56.766, E3 +53479.221}
SPL {X  -143.482, Y  +747.279, Z    +0.000, E1   -50.227, E3 +53497.234}
SPL {X  -154.118, Y  +719.449, Z    +0.000, E1   -38.836, E3 +53503.813}
SPL {X  -158.958, Y  +694.646, Z    +0.000, E1   -21.132, E3 +53506.664}
SPL {X  -159.960, Y  +679.609, Z    +0.000, E1    -6.021, E3 +53507.364}
SPL {X  -159.990, Y  +674.508, Z    +0.000, E1    -0.018, E3 +53507.423}
SPL {X  -159.990, Y  +672.787, Z    +0.000, E1    +4.022, E3 +53507.435}
SPL {X  -159.990, Y  +669.267, Z    +0.000, E1   +13.665, E3 +53507.505}
SPL {X  -159.990, Y  +663.438, Z    +0.000, E1   +29.379, E3 +53507.776}
SPL {X  -159.990, Y  +655.264, Z    +0.000, E1   +47.291, E3 +53508.393}
SPL {X  -159.990, Y  +645.368, Z    +0.000, E1   +59.257, E3 +53509.636}
SPL {X  -159.990, Y  +624.023, Z    +0.000, E1   +69.513, E3 +53513.761}
SPL {X  -159.990, Y  +543.075, Z    +0.000, E1   +75.590, E3 +53537.409}
SPL {X  -156.121, Y  +342.530, Z    +0.000, E1   +75.868, E3 +53624.055}
SPL {X  -153.498, Y  +332.386, Z    +0.000, E1   +75.628, E3 +53632.059}
ENDSPLINE

SPLINE
SPL {X  -155.252, Y  +338.851, Z    +0.000, E1   +74.632, E3 +53639.438}
SPL {X  -159.103, Y  +360.678, Z    +0.000, E1   +72.233, E3 +53651.763}
ENDSPLINE

SPLINE
SPL {X  -154.371, Y  +335.471, Z    +0.000, E1   +73.016, E3 +53660.333}
SPL {X  -149.938, Y  +321.685, Z    +0.000, E1   +73.398, E3 +53665.028}
SPL {X  -145.016, Y  +309.920, Z    +0.000, E1   +73.647, E3 +53669.549}
SPL {X  -139.138, Y  +298.522, Z    +0.000, E1   +74.138, E3 +53671.565}
SPL {X  -135.697, Y  +292.747, Z    +0.000, E1   +74.259, E3 +53673.566}
SPL {X  -132.590, Y  +287.964, Z    +0.000, E1   +73.910, E3 +53678.595}
SPL {X  -129.541, Y  +283.606, Z    +0.000, E1   +73.551, E3 +53683.235}
SPL {X  -126.457, Y  +279.493, Z    +0.000, E1   +73.175, E3 +53687.634}
SPL {X  -122.770, Y  +274.912, Z    +0.000, E1   +72.712, E3 +53692.489}
SPL {X  -119.156, Y  +270.736, Z    +0.000, E1   +72.213, E3 +53696.839}
SPL {X  -117.531, Y  +268.949, Z    +0.000, E1   +71.964, E3 +53698.654}
SPL {X   -74.907, Y  +236.129, Z    +0.000, E1   +61.720, E3 +53775.690}
ENDSPLINE

